LIN {X 0,Y 174.751,Z 590.29,A -85,B 0,C 180,E1 -20666.168,E2 -20666.168} C_VEL
LIN {X 0,Y 175.448,Z 592.178,A -85,B 0,C 180,E1 -20665.716,E2 -20665.716} C_VEL
LIN {X 0,Y 170.864,Z 646.273,A -85,B 0,C 180,E1 -20663.89,E2 -20663.89} C_VEL
LIN {X 0,Y 168.633,Z 660.424,A -85,B 0,C 180,E1 -20663.092,E2 -20663.092} C_VEL
LIN {X 0,Y 165.16,Z 674.762,A -85,B 0,C 180,E1 -20661.921,E2 -20661.921} C_VEL
LIN {X 0,Y 160.858,Z 688.251,A -85,B 0,C 180,E1 -20660.352,E2 -20660.352} C_VEL
LIN {X 0,Y 156.099,Z 700.216,A -85,B 0,C 180,E1 -20658.455,E2 -20658.455} C_VEL
LIN {X 0,Y 150.998,Z 711.144,A -85,B 0,C 180,E1 -20656.167,E2 -20656.167} C_VEL
LIN {X 0,Y 145.727,Z 721.318,A -85,B 0,C 180,E1 -20653.335,E2 -20653.335} C_VEL
LIN {X 0,Y 139.98,Z 731.094,A -85,B 0,C 180,E1 -20649.797,E2 -20649.797} C_VEL
LIN {X 0,Y 134.657,Z 739.228,A -85,B 0,C 180,E1 -20645.951,E2 -20645.951} C_VEL
LIN {X 0,Y 129.545,Z 746.964,A -85,B 0,C 180,E1 -20641.018,E2 -20641.018} C_VEL
LIN {X 0,Y 125.777,Z 752.256,A -85,B 0,C 180,E1 -20636.547,E2 -20636.547} C_VEL
LIN {X 0,Y 123.001,Z 756.514,A -85,B 0,C 180,E1 -20631.797,E2 -20631.797} C_VEL
LIN {X 0,Y 121.021,Z 759.832,A -85,B 0,C 180,E1 -20626.875,E2 -20626.875} C_VEL
LIN {X 0,Y 119.673,Z 762.879,A -85,B 0,C 180,E1 -20620.143,E2 -20620.143} C_VEL
LIN {X 0,Y 119.597,Z 764.442,A -85,B 0,C 180,E1 -20613.364,E2 -20613.364} C_VEL
LIN {X 0,Y 119.785,Z 764.659,A -85,B 0,C 180,E1 -20609.996,E2 -20609.996} C_VEL
LIN {X 0,Y 119.65,Z 764.459,A -85,B 0,C 180,E1 -20606.628,E2 -20606.628} C_VEL
LIN {X 0,Y 120.033,Z 762.933,A -85,B 0,C 180,E1 -20599.879,E2 -20599.879} C_VEL
LIN {X 0,Y 121.971,Z 759.942,A -85,B 0,C 180,E1 -20593.251,E2 -20593.251} C_VEL
LIN {X 0,Y 124.627,Z 756.694,A -85,B 0,C 180,E1 -20588.493,E2 -20588.493} C_VEL
LIN {X 0,Y 126.269,Z 755.1,A -85,B 0,C 180,E1 -20586.415,E2 -20586.415} C_VEL
LIN {X 0,Y 130.164,Z 758.008,A -85,B 0,C 180,E1 -20580.922,E2 -20580.922} C_VEL
LIN {X 0,Y 136.162,Z 760.226,A -85,B 0,C 180,E1 -20575.401,E2 -20575.401} C_VEL
LIN {X 0,Y 143.723,Z 761.469,A -85,B 0,C 180,E1 -20570.524,E2 -20570.524} C_VEL
LIN {X 0,Y 152.615,Z 761.755,A -85,B 0,C 180,E1 -20566.306,E2 -20566.306} C_VEL
LIN {X 0,Y 160.985,Z 761.235,A -85,B 0,C 180,E1 -20563.302,E2 -20563.302} C_VEL
LIN {X 0,Y 161.397,Z 761.087,A -85,B 0,C 180,E1 -20562.555,E2 -20562.555} C_VEL
LIN {X 0,Y 153.739,Z 760.626,A -85,B 0,C 180,E1 -20559.791,E2 -20559.791} C_VEL
LIN {X 0,Y 144.738,Z 758.979,A -85,B 0,C 180,E1 -20555.639,E2 -20555.639} C_VEL
LIN {X 0,Y 140.613,Z 757.696,A -85,B 0,C 180,E1 -20553.352,E2 -20553.352} C_VEL
LIN {X 0,Y 133.608,Z 754.257,A -85,B 0,C 180,E1 -20548.256,E2 -20548.256} C_VEL
LIN {X 0,Y 128.205,Z 749.58,A -85,B 0,C 180,E1 -20542.565,E2 -20542.565} C_VEL
LIN {X 0,Y 124.544,Z 743.565,A -85,B 0,C 180,E1 -20536.388,E2 -20536.388} C_VEL
LIN {X 0,Y 122.611,Z 737,A -85,B 0,C 180,E1 -20530.736,E2 -20530.736} C_VEL
LIN {X 0,Y 122.043,Z 729.036,A -85,B 0,C 180,E1 -20524.955,E2 -20524.955} C_VEL
LIN {X 0,Y 122.077,Z 720.491,A -85,B 0,C 180,E1 -20520,E2 -20520} C_VEL
LIN {X 0,Y 122.258,Z 711.841,A -85,B 0,C 180,E1 -20515.879,E2 -20515.879} C_VEL
LIN {X 0,Y 122.735,Z 702.53,A -85,B 0,C 180,E1 -20512.183,E2 -20512.183} C_VEL
LIN {X 0,Y 123.406,Z 691.305,A -85,B 0,C 180,E1 -20508.55,E2 -20508.55} C_VEL
LIN {X 0,Y 123.591,Z 689.165,A -85,B 0,C 180,E1 -20507.466,E2 -20507.466} C_VEL
LIN {X 0,Y 123.823,Z 687.977,A -85,B 0,C 180,E1 -20506.056,E2 -20506.056} C_VEL
LIN {X 0,Y 124.277,Z 687.395,A -85,B 0,C 180,E1 -20504.226,E2 -20504.226} C_VEL
LIN {X 0,Y 125.905,Z 686.979,A -85,B 0,C 180,E1 -20501.018,E2 -20501.018} C_VEL
LIN {X 0,Y 127.633,Z 685.962,A -85,B 0,C 180,E1 -20499.327,E2 -20499.327} C_VEL
LIN {X 0,Y 129.648,Z 684.696,A -85,B 0,C 180,E1 -20497.699,E2 -20497.699} C_VEL
LIN {X 0,Y 133.094,Z 681.626,A -85,B 0,C 180,E1 -20495.842,E2 -20495.842} C_VEL
LIN {X 0,Y 137.05,Z 677.069,A -85,B 0,C 180,E1 -20494.334,E2 -20494.334} C_VEL
LIN {X 0,Y 138.247,Z 675.526,A -85,B 0,C 180,E1 -20493.975,E2 -20493.975} C_VEL
LIN {X 0,Y 141.117,Z 673.06,A -85,B 0,C 180,E1 -20492.488,E2 -20492.488} C_VEL
LIN {X 0,Y 145.003,Z 668.739,A -85,B 0,C 180,E1 -20491.008,E2 -20491.008} C_VEL
LIN {X 0,Y 149.365,Z 662.342,A -85,B 0,C 180,E1 -20489.788,E2 -20489.788} C_VEL
LIN {X 0,Y 153.704,Z 653.819,A -85,B 0,C 180,E1 -20488.901,E2 -20488.901} C_VEL
LIN {X 0,Y 154.898,Z 651.2,A -85,B 0,C 180,E1 -20488.661,E2 -20488.661} C_VEL
LIN {X 0,Y 158.174,Z 646.403,A -85,B 0,C 180,E1 -20487.439,E2 -20487.439} C_VEL
LIN {X 0,Y 161.889,Z 638.911,A -85,B 0,C 180,E1 -20486.261,E2 -20486.261} C_VEL
LIN {X 0,Y 165.983,Z 627.33,A -85,B 0,C 180,E1 -20485.022,E2 -20485.022} C_VEL
LIN {X 0,Y 169.425,Z 615.622,A -85,B 0,C 180,E1 -20484.131,E2 -20484.131} C_VEL
LIN {X 0,Y 167.38,Z 640.416,A -85,B 0,C 180,E1 -20483.235,E2 -20483.235} C_VEL
LIN {X 0,Y 165.141,Z 654.079,A -85,B 0,C 180,E1 -20482.437,E2 -20482.437} C_VEL
LIN {X 0,Y 162.14,Z 666.874,A -85,B 0,C 180,E1 -20481.285,E2 -20481.285} C_VEL
LIN {X 0,Y 157.903,Z 680.096,A -85,B 0,C 180,E1 -20479.664,E2 -20479.664} C_VEL
LIN {X 0,Y 153.219,Z 691.732,A -85,B 0,C 180,E1 -20477.705,E2 -20477.705} C_VEL
LIN {X 0,Y 148.082,Z 702.301,A -85,B 0,C 180,E1 -20475.394,E2 -20475.394} C_VEL
LIN {X 0,Y 142.637,Z 712.201,A -85,B 0,C 180,E1 -20472.492,E2 -20472.492} C_VEL
LIN {X 0,Y 136.949,Z 721.337,A -85,B 0,C 180,E1 -20468.955,E2 -20468.955} C_VEL
LIN {X 0,Y 131.412,Z 728.995,A -85,B 0,C 180,E1 -20465.098,E2 -20465.098} C_VEL
LIN {X 0,Y 125.818,Z 736.115,A -85,B 0,C 180,E1 -20460.185,E2 -20460.185} C_VEL
LIN {X 0,Y 121.759,Z 740.971,A -85,B 0,C 180,E1 -20455.657,E2 -20455.657} C_VEL
LIN {X 0,Y 118.435,Z 744.801,A -85,B 0,C 180,E1 -20450.862,E2 -20450.862} C_VEL
LIN {X 0,Y 115.262,Z 748.408,A -85,B 0,C 180,E1 -20444.121,E2 -20444.121} C_VEL
LIN {X 0,Y 113.482,Z 750.529,A -85,B 0,C 180,E1 -20437.12,E2 -20437.12} C_VEL
LIN {X 0,Y 112.893,Z 751.232,A -85,B 0,C 180,E1 -20430.005,E2 -20430.005} C_VEL
LIN {X 0,Y 113.479,Z 750.486,A -85,B 0,C 180,E1 -20422.89,E2 -20422.89} C_VEL
LIN {X 0,Y 115.257,Z 748.33,A -85,B 0,C 180,E1 -20415.888,E2 -20415.888} C_VEL
LIN {X 0,Y 118.436,Z 744.678,A -85,B 0,C 180,E1 -20409.148,E2 -20409.148} C_VEL
LIN {X 0,Y 121.806,Z 740.807,A -85,B 0,C 180,E1 -20404.364,E2 -20404.364} C_VEL
LIN {X 0,Y 125.949,Z 735.902,A -85,B 0,C 180,E1 -20399.859,E2 -20399.859} C_VEL
LIN {X 0,Y 130.592,Z 729.843,A -85,B 0,C 180,E1 -20395.598,E2 -20395.598} C_VEL
LIN {X 0,Y 136.018,Z 722.398,A -85,B 0,C 180,E1 -20391.687,E2 -20391.687} C_VEL
LIN {X 0,Y 141.435,Z 713.947,A -85,B 0,C 180,E1 -20388.264,E2 -20388.264} C_VEL
LIN {X 0,Y 147.09,Z 703.928,A -85,B 0,C 180,E1 -20385.195,E2 -20385.195} C_VEL
LIN {X 0,Y 152.145,Z 693.71,A -85,B 0,C 180,E1 -20382.841,E2 -20382.841} C_VEL
LIN {X 0,Y 156.789,Z 682.529,A -85,B 0,C 180,E1 -20380.857,E2 -20380.857} C_VEL
LIN {X 0,Y 160.982,Z 670.126,A -85,B 0,C 180,E1 -20379.209,E2 -20379.209} C_VEL
LIN {X 0,Y 164.303,Z 657.215,A -85,B 0,C 180,E1 -20377.946,E2 -20377.946} C_VEL
LIN {X 0,Y 166.571,Z 644.664,A -85,B 0,C 180,E1 -20377.095,E2 -20377.095} C_VEL
LIN {X 0,Y 168.055,Z 630.758,A -85,B 0,C 180,E1 -20376.513,E2 -20376.513} C_VEL
LIN {X 0,Y 171.047,Z 593.041,A -85,B 0,C 180,E1 -20375.296,E2 -20375.296} C_VEL
LIN {X 0,Y 167.73,Z 584.739,A -85,B 0,C 180,E1 -20372.916,E2 -20372.916} C_VEL
LIN {X 0,Y 163.421,Z 575.531,A -85,B 0,C 180,E1 -20369.525,E2 -20369.525} C_VEL
LIN {X 0,Y 160.098,Z 569.15,A -85,B 0,C 180,E1 -20366.549,E2 -20366.549} C_VEL
LIN {X 0,Y 156.776,Z 563.254,A -85,B 0,C 180,E1 -20363.109,E2 -20363.109} C_VEL
LIN {X 0,Y 153.307,Z 557.682,A -85,B 0,C 180,E1 -20358.718,E2 -20358.718} C_VEL
LIN {X 0,Y 150.18,Z 552.762,A -85,B 0,C 180,E1 -20353.188,E2 -20353.188} C_VEL
LIN {X 0,Y 147.985,Z 549.73,A -85,B 0,C 180,E1 -20346.3,E2 -20346.3} C_VEL
LIN {X 0,Y 147.618,Z 548.691,A -85,B 0,C 180,E1 -20341.345,E2 -20341.345} C_VEL
LIN {X 0,Y 147.76,Z 549.144,A -85,B 0,C 180,E1 -20338.638,E2 -20338.638} C_VEL
LIN {X 0,Y 149.497,Z 552.083,A -85,B 0,C 180,E1 -20331.538,E2 -20331.538} C_VEL
LIN {X 0,Y 150.744,Z 553.976,A -85,B 0,C 180,E1 -20328.742,E2 -20328.742} C_VEL
LIN {X 0,Y 154.198,Z 559.575,A -85,B 0,C 180,E1 -20323.149,E2 -20323.149} C_VEL
LIN {X 0,Y 157.289,Z 564.846,A -85,B 0,C 180,E1 -20319.38,E2 -20319.38} C_VEL
LIN {X 0,Y 160.115,Z 570.007,A -85,B 0,C 180,E1 -20316.475,E2 -20316.475} C_VEL
LIN {X 0,Y 163.501,Z 576.58,A -85,B 0,C 180,E1 -20313.429,E2 -20313.429} C_VEL
LIN {X 0,Y 167.808,Z 586.127,A -85,B 0,C 180,E1 -20310.003,E2 -20310.003} C_VEL
LIN {X 0,Y 171.157,Z 594.739,A -85,B 0,C 180,E1 -20307.564,E2 -20307.564} C_VEL
LIN {X 0,Y 166.751,Z 645.455,A -85,B 0,C 180,E1 -20305.842,E2 -20305.842} C_VEL
LIN {X 0,Y 164.492,Z 659.477,A -85,B 0,C 180,E1 -20305.092,E2 -20305.092} C_VEL
LIN {X 0,Y 161.167,Z 673,A -85,B 0,C 180,E1 -20304.036,E2 -20304.036} C_VEL
LIN {X 0,Y 157.033,Z 685.93,A -85,B 0,C 180,E1 -20302.592,E2 -20302.592} C_VEL
LIN {X 0,Y 152.067,Z 698.358,A -85,B 0,C 180,E1 -20300.72,E2 -20300.72} C_VEL
LIN {X 0,Y 146.705,Z 709.591,A -85,B 0,C 180,E1 -20298.457,E2 -20298.457} C_VEL
LIN {X 0,Y 141.085,Z 720.013,A -85,B 0,C 180,E1 -20295.62,E2 -20295.62} C_VEL
LIN {X 0,Y 135.553,Z 729.147,A -85,B 0,C 180,E1 -20292.371,E2 -20292.371} C_VEL
LIN {X 0,Y 129.818,Z 737.545,A -85,B 0,C 180,E1 -20288.499,E2 -20288.499} C_VEL
LIN {X 0,Y 124.139,Z 745.513,A -85,B 0,C 180,E1 -20283.498,E2 -20283.498} C_VEL
LIN {X 0,Y 119.214,Z 752.093,A -85,B 0,C 180,E1 -20277.836,E2 -20277.836} C_VEL
LIN {X 0,Y 115.577,Z 757.318,A -85,B 0,C 180,E1 -20271.393,E2 -20271.393} C_VEL
LIN {X 0,Y 113.214,Z 761.13,A -85,B 0,C 180,E1 -20264.373,E2 -20264.373} C_VEL
LIN {X 0,Y 112.407,Z 763.432,A -85,B 0,C 180,E1 -20257.179,E2 -20257.179} C_VEL
LIN {X 0,Y 112.541,Z 764.134,A -85,B 0,C 180,E1 -20252.333,E2 -20252.333} C_VEL
LIN {X 0,Y 112.691,Z 764.25,A -85,B 0,C 180,E1 -20249.995,E2 -20249.995} C_VEL
LIN {X 0,Y 112.555,Z 764.049,A -85,B 0,C 180,E1 -20246.415,E2 -20246.415} C_VEL
LIN {X 0,Y 112.66,Z 763.47,A -85,B 0,C 180,E1 -20242.828,E2 -20242.828} C_VEL
LIN {X 0,Y 113.903,Z 761.214,A -85,B 0,C 180,E1 -20235.707,E2 -20235.707} C_VEL
LIN {X 0,Y 116.945,Z 757.47,A -85,B 0,C 180,E1 -20228.86,E2 -20228.86} C_VEL
LIN {X 0,Y 120.851,Z 753.596,A -85,B 0,C 180,E1 -20223.905,E2 -20223.905} C_VEL
LIN {X 0,Y 127.135,Z 757.49,A -85,B 0,C 180,E1 -20216.436,E2 -20216.436} C_VEL
LIN {X 0,Y 134.293,Z 759.63,A -85,B 0,C 180,E1 -20211.093,E2 -20211.093} C_VEL
LIN {X 0,Y 142.821,Z 760.817,A -85,B 0,C 180,E1 -20206.451,E2 -20206.451} C_VEL
LIN {X 0,Y 150.668,Z 761.111,A -85,B 0,C 180,E1 -20203.268,E2 -20203.268} C_VEL
LIN {X 0,Y 150.095,Z 760.873,A -85,B 0,C 180,E1 -20202.206,E2 -20202.206} C_VEL
LIN {X 0,Y 143.541,Z 759.697,A -85,B 0,C 180,E1 -20199.531,E2 -20199.531} C_VEL
LIN {X 0,Y 134.792,Z 756.968,A -85,B 0,C 180,E1 -20194.997,E2 -20194.997} C_VEL
LIN {X 0,Y 127.504,Z 753.065,A -85,B 0,C 180,E1 -20189.741,E2 -20189.741} C_VEL
LIN {X 0,Y 121.857,Z 747.927,A -85,B 0,C 180,E1 -20183.811,E2 -20183.811} C_VEL
LIN {X 0,Y 118.049,Z 741.477,A -85,B 0,C 180,E1 -20177.317,E2 -20177.317} C_VEL
LIN {X 0,Y 115.897,Z 733.429,A -85,B 0,C 180,E1 -20170.481,E2 -20170.481} C_VEL
LIN {X 0,Y 115.491,Z 726.032,A -85,B 0,C 180,E1 -20165.237,E2 -20165.237} C_VEL
LIN {X 0,Y 115.449,Z 718.689,A -85,B 0,C 180,E1 -20160.871,E2 -20160.871} C_VEL
LIN {X 0,Y 115.657,Z 708.699,A -85,B 0,C 180,E1 -20156.08,E2 -20156.08} C_VEL
LIN {X 0,Y 116.092,Z 698.828,A -85,B 0,C 180,E1 -20152.171,E2 -20152.171} C_VEL
LIN {X 0,Y 116.215,Z 695.374,A -85,B 0,C 180,E1 -20150.92,E2 -20150.92} C_VEL
LIN {X 0,Y 115.98,Z 695.896,A -85,B 0,C 180,E1 -20150.407,E2 -20150.407} C_VEL
LIN {X 0,Y 116.047,Z 696.135,A -85,B 0,C 180,E1 -20149.532,E2 -20149.532} C_VEL
LIN {X 0,Y 117.022,Z 695.467,A -85,B 0,C 180,E1 -20147.865,E2 -20147.865} C_VEL
LIN {X 0,Y 120.501,Z 692.137,A -85,B 0,C 180,E1 -20144.784,E2 -20144.784} C_VEL
LIN {X 0,Y 123.407,Z 690.151,A -85,B 0,C 180,E1 -20141.746,E2 -20141.746} C_VEL
LIN {X 0,Y 125.691,Z 687.944,A -85,B 0,C 180,E1 -20140.397,E2 -20140.397} C_VEL
LIN {X 0,Y 127.127,Z 686.36,A -85,B 0,C 180,E1 -20139.702,E2 -20139.702} C_VEL
LIN {X 0,Y 127.633,Z 685.962,A -85,B 0,C 180,E1 -20139.327,E2 -20139.327} C_VEL
LIN {X 0,Y 130.12,Z 684.459,A -85,B 0,C 180,E1 -20137.326,E2 -20137.326} C_VEL
LIN {X 0,Y 135.875,Z 682.058,A -85,B 0,C 180,E1 -20132.88,E2 -20132.88} C_VEL
LIN {X 0,Y 138.121,Z 680.497,A -85,B 0,C 180,E1 -20131.678,E2 -20131.678} C_VEL
LIN {X 0,Y 142.493,Z 676.654,A -85,B 0,C 180,E1 -20129.897,E2 -20129.897} C_VEL
LIN {X 0,Y 145.897,Z 673.011,A -85,B 0,C 180,E1 -20128.812,E2 -20128.812} C_VEL
LIN {X 0,Y 150.887,Z 666.322,A -85,B 0,C 180,E1 -20127.613,E2 -20127.613} C_VEL
LIN {X 0,Y 155.631,Z 657.999,A -85,B 0,C 180,E1 -20126.796,E2 -20126.796} C_VEL
LIN {X 0,Y 157.05,Z 655.124,A -85,B 0,C 180,E1 -20126.542,E2 -20126.542} C_VEL
LIN {X 0,Y 160.655,Z 649.982,A -85,B 0,C 180,E1 -20125.432,E2 -20125.432} C_VEL
LIN {X 0,Y 162.342,Z 647.1,A -85,B 0,C 180,E1 -20124.961,E2 -20124.961} C_VEL
LIN {X 0,Y 159.457,Z 661.267,A -85,B 0,C 180,E1 -20123.903,E2 -20123.903} C_VEL
LIN {X 0,Y 155.953,Z 673.577,A -85,B 0,C 180,E1 -20122.591,E2 -20122.591} C_VEL
LIN {X 0,Y 151.65,Z 685.301,A -85,B 0,C 180,E1 -20120.924,E2 -20120.924} C_VEL
LIN {X 0,Y 146.125,Z 697.171,A -85,B 0,C 180,E1 -20118.725,E2 -20118.725} C_VEL
LIN {X 0,Y 140.912,Z 706.825,A -85,B 0,C 180,E1 -20116.323,E2 -20116.323} C_VEL
LIN {X 0,Y 135.252,Z 716.191,A -85,B 0,C 180,E1 -20113.203,E2 -20113.203} C_VEL
LIN {X 0,Y 129.513,Z 724.461,A -85,B 0,C 180,E1 -20109.619,E2 -20109.619} C_VEL
LIN {X 0,Y 123.922,Z 731.606,A -85,B 0,C 180,E1 -20105.547,E2 -20105.547} C_VEL
LIN {X 0,Y 118.24,Z 738.292,A -85,B 0,C 180,E1 -20100.351,E2 -20100.351} C_VEL
LIN {X 0,Y 114.142,Z 742.772,A -85,B 0,C 180,E1 -20095.536,E2 -20095.536} C_VEL
LIN {X 0,Y 111.84,Z 745.21,A -85,B 0,C 180,E1 -20092.155,E2 -20092.155} C_VEL
LIN {X 0,Y 108.391,Z 748.817,A -85,B 0,C 180,E1 -20085.037,E2 -20085.037} C_VEL
LIN {X 0,Y 106.463,Z 750.937,A -85,B 0,C 180,E1 -20077.592,E2 -20077.592} C_VEL
LIN {X 0,Y 105.824,Z 751.64,A -85,B 0,C 180,E1 -20070.005,E2 -20070.005} C_VEL
LIN {X 0,Y 106.461,Z 750.894,A -85,B 0,C 180,E1 -20062.418,E2 -20062.418} C_VEL
LIN {X 0,Y 108.385,Z 748.74,A -85,B 0,C 180,E1 -20054.972,E2 -20054.972} C_VEL
LIN {X 0,Y 111.841,Z 745.089,A -85,B 0,C 180,E1 -20047.855,E2 -20047.855} C_VEL
LIN {X 0,Y 115.461,Z 741.218,A -85,B 0,C 180,E1 -20042.843,E2 -20042.843} C_VEL
LIN {X 0,Y 119.858,Z 736.318,A -85,B 0,C 180,E1 -20038.154,E2 -20038.154} C_VEL
LIN {X 0,Y 124.818,Z 730.262,A -85,B 0,C 180,E1 -20033.762,E2 -20033.762} C_VEL
LIN {X 0,Y 130.541,Z 722.824,A -85,B 0,C 180,E1 -20029.761,E2 -20029.761} C_VEL
LIN {X 0,Y 136.559,Z 713.876,A -85,B 0,C 180,E1 -20026.097,E2 -20026.097} C_VEL
LIN {X 0,Y 142.147,Z 704.392,A -85,B 0,C 180,E1 -20023.181,E2 -20023.181} C_VEL
LIN {X 0,Y 147.434,Z 694.197,A -85,B 0,C 180,E1 -20020.828,E2 -20020.828} C_VEL
LIN {X 0,Y 152.259,Z 683.054,A -85,B 0,C 180,E1 -20018.845,E2 -20018.845} C_VEL
LIN {X 0,Y 156.615,Z 670.711,A -85,B 0,C 180,E1 -20017.207,E2 -20017.207} C_VEL
LIN {X 0,Y 160.061,Z 657.901,A -85,B 0,C 180,E1 -20015.954,E2 -20015.954} C_VEL
LIN {X 0,Y 162.412,Z 645.601,A -85,B 0,C 180,E1 -20015.109,E2 -20015.109} C_VEL
LIN {X 0,Y 163.958,Z 632.23,A -85,B 0,C 180,E1 -20014.533,E2 -20014.533} C_VEL
LIN {X 0,Y 166.984,Z 595.617,A -85,B 0,C 180,E1 -20013.352,E2 -20013.352} C_VEL
LIN {X 0,Y 163.154,Z 586.222,A -85,B 0,C 180,E1 -20010.301,E2 -20010.301} C_VEL
LIN {X 0,Y 159.55,Z 578.432,A -85,B 0,C 180,E1 -20007.075,E2 -20007.075} C_VEL
LIN {X 0,Y 156.34,Z 572.241,A -85,B 0,C 180,E1 -20003.779,E2 -20003.779} C_VEL
LIN {X 0,Y 153.865,Z 567.749,A -85,B 0,C 180,E1 -20000.803,E2 -20000.803} C_VEL
LIN {X 0,Y 151.679,Z 564.144,A -85,B 0,C 180,E1 -19997.703,E2 -19997.703} C_VEL
LIN {X 0,Y 149.018,Z 559.587,A -85,B 0,C 180,E1 -19992.599,E2 -19992.599} C_VEL
LIN {X 0,Y 147.106,Z 556.814,A -85,B 0,C 180,E1 -19986.258,E2 -19986.258} C_VEL
LIN {X 0,Y 146.748,Z 556.001,A -85,B 0,C 180,E1 -19982.745,E2 -19982.745} C_VEL
LIN {X 0,Y 146.814,Z 555.905,A -85,B 0,C 180,E1 -19979.658,E2 -19979.658} C_VEL
LIN {X 0,Y 148.364,Z 558.901,A -85,B 0,C 180,E1 -19972.173,E2 -19972.173} C_VEL
LIN {X 0,Y 149.535,Z 560.838,A -85,B 0,C 180,E1 -19969.336,E2 -19969.336} C_VEL
LIN {X 0,Y 152.627,Z 566.192,A -85,B 0,C 180,E1 -19963.962,E2 -19963.962} C_VEL
LIN {X 0,Y 155.328,Z 571.036,A -85,B 0,C 180,E1 -19960.422,E2 -19960.422} C_VEL
LIN {X 0,Y 158.322,Z 576.818,A -85,B 0,C 180,E1 -19957.144,E2 -19957.144} C_VEL
LIN {X 0,Y 161.296,Z 583.175,A -85,B 0,C 180,E1 -19954.285,E2 -19954.285} C_VEL
LIN {X 0,Y 164.848,Z 591.51,A -85,B 0,C 180,E1 -19951.25,E2 -19951.25} C_VEL
LIN {X 0,Y 167.045,Z 597.374,A -85,B 0,C 180,E1 -19949.503,E2 -19949.503} C_VEL
LIN {X 0,Y 162.682,Z 645.77,A -85,B 0,C 180,E1 -19947.858,E2 -19947.858} C_VEL
LIN {X 0,Y 160.301,Z 659.728,A -85,B 0,C 180,E1 -19947.108,E2 -19947.108} C_VEL
LIN {X 0,Y 156.757,Z 673.502,A -85,B 0,C 180,E1 -19946.033,E2 -19946.033} C_VEL
LIN {X 0,Y 152.808,Z 685.375,A -85,B 0,C 180,E1 -19944.716,E2 -19944.716} C_VEL
LIN {X 0,Y 147.658,Z 697.849,A -85,B 0,C 180,E1 -19942.861,E2 -19942.861} C_VEL
LIN {X 0,Y 142.094,Z 709.123,A -85,B 0,C 180,E1 -19940.601,E2 -19940.601} C_VEL
LIN {X 0,Y 136.6,Z 718.82,A -85,B 0,C 180,E1 -19938.023,E2 -19938.023} C_VEL
LIN {X 0,Y 130.345,Z 728.71,A -85,B 0,C 180,E1 -19934.496,E2 -19934.496} C_VEL
LIN {X 0,Y 124.307,Z 737.117,A -85,B 0,C 180,E1 -19930.549,E2 -19930.549} C_VEL
LIN {X 0,Y 118.219,Z 745.089,A -85,B 0,C 180,E1 -19925.418,E2 -19925.418} C_VEL
LIN {X 0,Y 113.151,Z 751.418,A -85,B 0,C 180,E1 -19919.789,E2 -19919.789} C_VEL
LIN {X 0,Y 109.799,Z 755.68,A -85,B 0,C 180,E1 -19914.58,E2 -19914.58} C_VEL
LIN {X 0,Y 107.391,Z 759.003,A -85,B 0,C 180,E1 -19909.095,E2 -19909.095} C_VEL
LIN {X 0,Y 105.623,Z 762.053,A -85,B 0,C 180,E1 -19901.509,E2 -19901.509} C_VEL
LIN {X 0,Y 105.391,Z 763.62,A -85,B 0,C 180,E1 -19893.819,E2 -19893.819} C_VEL
LIN {X 0,Y 105.597,Z 763.84,A -85,B 0,C 180,E1 -19889.995,E2 -19889.995} C_VEL
LIN {X 0,Y 105.463,Z 763.639,A -85,B 0,C 180,E1 -19886.174,E2 -19886.174} C_VEL
LIN {X 0,Y 105.606,Z 763.06,A -85,B 0,C 180,E1 -19882.346,E2 -19882.346} C_VEL
LIN {X 0,Y 107.01,Z 760.803,A -85,B 0,C 180,E1 -19874.764,E2 -19874.764} C_VEL
LIN {X 0,Y 110.344,Z 757.059,A -85,B 0,C 180,E1 -19867.528,E2 -19867.528} C_VEL
LIN {X 0,Y 115.494,Z 752.104,A -85,B 0,C 180,E1 -19861.361,E2 -19861.361} C_VEL
LIN {X 0,Y 115.877,Z 752.058,A -85,B 0,C 180,E1 -19860.969,E2 -19860.969} C_VEL
LIN {X 0,Y 121.511,Z 755.529,A -85,B 0,C 180,E1 -19854.658,E2 -19854.658} C_VEL
LIN {X 0,Y 128.981,Z 758.069,A -85,B 0,C 180,E1 -19849.162,E2 -19849.162} C_VEL
LIN {X 0,Y 139.647,Z 759.866,A -85,B 0,C 180,E1 -19843.665,E2 -19843.665} C_VEL
LIN {X 0,Y 140.607,Z 759.968,A -85,B 0,C 180,E1 -19843.271,E2 -19843.271} C_VEL
LIN {X 0,Y 139.919,Z 759.638,A -85,B 0,C 180,E1 -19842.147,E2 -19842.147} C_VEL
LIN {X 0,Y 133.521,Z 757.741,A -85,B 0,C 180,E1 -19839.17,E2 -19839.17} C_VEL
LIN {X 0,Y 125.179,Z 753.97,A -85,B 0,C 180,E1 -19834.155,E2 -19834.155} C_VEL
LIN {X 0,Y 118.379,Z 749.006,A -85,B 0,C 180,E1 -19828.356,E2 -19828.356} C_VEL
LIN {X 0,Y 113.418,Z 742.771,A -85,B 0,C 180,E1 -19821.826,E2 -19821.826} C_VEL
LIN {X 0,Y 110.584,Z 736.136,A -85,B 0,C 180,E1 -19815.67,E2 -19815.67} C_VEL
LIN {X 0,Y 109.179,Z 726.907,A -85,B 0,C 180,E1 -19808.327,E2 -19808.327} C_VEL
LIN {X 0,Y 108.962,Z 718.206,A -85,B 0,C 180,E1 -19802.772,E2 -19802.772} C_VEL
LIN {X 0,Y 109.001,Z 709.366,A -85,B 0,C 180,E1 -19798.152,E2 -19798.152} C_VEL
LIN {X 0,Y 109.105,Z 704.328,A -85,B 0,C 180,E1 -19795.844,E2 -19795.844} C_VEL
LIN {X 0,Y 108.732,Z 704.907,A -85,B 0,C 180,E1 -19794.436,E2 -19794.436} C_VEL
LIN {X 0,Y 109.327,Z 704.436,A -85,B 0,C 180,E1 -19792.613,E2 -19792.613} C_VEL
LIN {X 0,Y 111.986,Z 701.907,A -85,B 0,C 180,E1 -19789.147,E2 -19789.147} C_VEL
LIN {X 0,Y 114.256,Z 700.43,A -85,B 0,C 180,E1 -19785.756,E2 -19785.756} C_VEL
LIN {X 0,Y 117.495,Z 697.696,A -85,B 0,C 180,E1 -19783.159,E2 -19783.159} C_VEL
LIN {X 0,Y 121.319,Z 695.24,A -85,B 0,C 180,E1 -19779.66,E2 -19779.66} C_VEL
LIN {X 0,Y 126.155,Z 691.085,A -85,B 0,C 180,E1 -19777.047,E2 -19777.047} C_VEL
LIN {X 0,Y 128.083,Z 689.921,A -85,B 0,C 180,E1 -19775.698,E2 -19775.698} C_VEL
LIN {X 0,Y 132.275,Z 686.527,A -85,B 0,C 180,E1 -19773.668,E2 -19773.668} C_VEL
LIN {X 0,Y 136.085,Z 682.702,A -85,B 0,C 180,E1 -19772.302,E2 -19772.302} C_VEL
LIN {X 0,Y 138.121,Z 680.497,A -85,B 0,C 180,E1 -19771.678,E2 -19771.678} C_VEL
LIN {X 0,Y 141.302,Z 678.49,A -85,B 0,C 180,E1 -19770.035,E2 -19770.035} C_VEL
LIN {X 0,Y 146.87,Z 675.936,A -85,B 0,C 180,E1 -19767.119,E2 -19767.119} C_VEL
LIN {X 0,Y 149.751,Z 673.72,A -85,B 0,C 180,E1 -19766.042,E2 -19766.042} C_VEL
LIN {X 0,Y 150.936,Z 672.387,A -85,B 0,C 180,E1 -19765.742,E2 -19765.742} C_VEL
LIN {X 0,Y 152.462,Z 670.362,A -85,B 0,C 180,E1 -19765.463,E2 -19765.463} C_VEL
LIN {X 0,Y 152.39,Z 672.172,A -85,B 0,C 180,E1 -19764.95,E2 -19764.95} C_VEL
LIN {X 0,Y 147.914,Z 684.265,A -85,B 0,C 180,E1 -19763.307,E2 -19763.307} C_VEL
LIN {X 0,Y 142.819,Z 695.255,A -85,B 0,C 180,E1 -19761.375,E2 -19761.375} C_VEL
LIN {X 0,Y 137.323,Z 705.322,A -85,B 0,C 180,E1 -19759.021,E2 -19759.021} C_VEL
LIN {X 0,Y 131.379,Z 714.847,A -85,B 0,C 180,E1 -19756.018,E2 -19756.018} C_VEL
LIN {X 0,Y 125.18,Z 723.549,A -85,B 0,C 180,E1 -19752.36,E2 -19752.36} C_VEL
LIN {X 0,Y 119.138,Z 730.928,A -85,B 0,C 180,E1 -19748.277,E2 -19748.277} C_VEL
LIN {X 0,Y 113.767,Z 736.941,A -85,B 0,C 180,E1 -19743.783,E2 -19743.783} C_VEL
LIN {X 0,Y 109.17,Z 741.79,A -85,B 0,C 180,E1 -19738.875,E2 -19738.875} C_VEL
LIN {X 0,Y 105.317,Z 745.618,A -85,B 0,C 180,E1 -19733.608,E2 -19733.608} C_VEL
LIN {X 0,Y 101.569,Z 749.225,A -85,B 0,C 180,E1 -19726.073,E2 -19726.073} C_VEL
LIN {X 0,Y 99.438,Z 751.346,A -85,B 0,C 180,E1 -19718.131,E2 -19718.131} C_VEL
LIN {X 0,Y 98.736,Z 752.049,A -85,B 0,C 180,E1 -19710.005,E2 -19710.005} C_VEL
LIN {X 0,Y 99.434,Z 751.304,A -85,B 0,C 180,E1 -19701.879,E2 -19701.879} C_VEL
LIN {X 0,Y 101.563,Z 749.149,A -85,B 0,C 180,E1 -19693.937,E2 -19693.937} C_VEL
LIN {X 0,Y 105.317,Z 745.499,A -85,B 0,C 180,E1 -19686.403,E2 -19686.403} C_VEL
LIN {X 0,Y 109.211,Z 741.629,A -85,B 0,C 180,E1 -19681.148,E2 -19681.148} C_VEL
LIN {X 0,Y 113.886,Z 736.734,A -85,B 0,C 180,E1 -19676.268,E2 -19676.268} C_VEL
LIN {X 0,Y 119.186,Z 730.681,A -85,B 0,C 180,E1 -19671.752,E2 -19671.752} C_VEL
LIN {X 0,Y 125.213,Z 723.251,A -85,B 0,C 180,E1 -19667.665,E2 -19667.665} C_VEL
LIN {X 0,Y 131.675,Z 714.102,A -85,B 0,C 180,E1 -19663.875,E2 -19663.875} C_VEL
LIN {X 0,Y 138.001,Z 703.795,A -85,B 0,C 180,E1 -19660.759,E2 -19660.759} C_VEL
LIN {X 0,Y 143.531,Z 693.404,A -85,B 0,C 180,E1 -19658.43,E2 -19658.43} C_VEL
LIN {X 0,Y 148.589,Z 682.005,A -85,B 0,C 180,E1 -19656.486,E2 -19656.486} C_VEL
LIN {X 0,Y 153.107,Z 669.308,A -85,B 0,C 180,E1 -19654.871,E2 -19654.871} C_VEL
LIN {X 0,Y 156.579,Z 656.024,A -85,B 0,C 180,E1 -19653.638,E2 -19653.638} C_VEL
LIN {X 0,Y 159.071,Z 642.186,A -85,B 0,C 180,E1 -19652.79,E2 -19652.79} C_VEL
LIN {X 0,Y 161.35,Z 619.119,A -85,B 0,C 180,E1 -19652.003,E2 -19652.003} C_VEL
LIN {X 0,Y 163.093,Z 598.441,A -85,B 0,C 180,E1 -19651.319,E2 -19651.319} C_VEL
LIN {X 0,Y 159.218,Z 588.732,A -85,B 0,C 180,E1 -19647.854,E2 -19647.854} C_VEL
LIN {X 0,Y 156.05,Z 581.76,A -85,B 0,C 180,E1 -19644.62,E2 -19644.62} C_VEL
LIN {X 0,Y 153.734,Z 577.167,A -85,B 0,C 180,E1 -19641.918,E2 -19641.918} C_VEL
LIN {X 0,Y 151.955,Z 573.777,A -85,B 0,C 180,E1 -19639.537,E2 -19639.537} C_VEL
LIN {X 0,Y 150.205,Z 570.703,A -85,B 0,C 180,E1 -19636.829,E2 -19636.829} C_VEL
LIN {X 0,Y 147.871,Z 566.432,A -85,B 0,C 180,E1 -19632.002,E2 -19632.002} C_VEL
LIN {X 0,Y 146.116,Z 563.7,A -85,B 0,C 180,E1 -19625.521,E2 -19625.521} C_VEL
LIN {X 0,Y 145.879,Z 563.086,A -85,B 0,C 180,E1 -19622.762,E2 -19622.762} C_VEL
LIN {X 0,Y 145.943,Z 563.002,A -85,B 0,C 180,E1 -19619.656,E2 -19619.656} C_VEL
LIN {X 0,Y 147.256,Z 565.724,A -85,B 0,C 180,E1 -19612.803,E2 -19612.803} C_VEL
LIN {X 0,Y 148.273,Z 567.537,A -85,B 0,C 180,E1 -19610.108,E2 -19610.108} C_VEL
LIN {X 0,Y 151.117,Z 572.839,A -85,B 0,C 180,E1 -19604.749,E2 -19604.749} C_VEL
LIN {X 0,Y 153.432,Z 577.289,A -85,B 0,C 180,E1 -19601.472,E2 -19601.472} C_VEL
LIN {X 0,Y 156.12,Z 582.807,A -85,B 0,C 180,E1 -19598.286,E2 -19598.286} C_VEL
LIN {X 0,Y 158.958,Z 589.288,A -85,B 0,C 180,E1 -19595.338,E2 -19595.338} C_VEL
LIN {X 0,Y 162.134,Z 597.32,A -85,B 0,C 180,E1 -19592.402,E2 -19592.402} C_VEL
LIN {X 0,Y 163.163,Z 600.213,A -85,B 0,C 180,E1 -19591.503,E2 -19591.503} C_VEL
LIN {X 0,Y 158.816,Z 646.037,A -85,B 0,C 180,E1 -19589.977,E2 -19589.977} C_VEL
LIN {X 0,Y 156.243,Z 660.344,A -85,B 0,C 180,E1 -19589.202,E2 -19589.202} C_VEL
LIN {X 0,Y 152.551,Z 674.005,A -85,B 0,C 180,E1 -19588.14,E2 -19588.14} C_VEL
LIN {X 0,Y 148.13,Z 686.593,A -85,B 0,C 180,E1 -19586.735,E2 -19586.735} C_VEL
LIN {X 0,Y 142.821,Z 698.741,A -85,B 0,C 180,E1 -19584.887,E2 -19584.887} C_VEL
LIN {X 0,Y 137.038,Z 709.745,A -85,B 0,C 180,E1 -19582.64,E2 -19582.64} C_VEL
LIN {X 0,Y 130.475,Z 720.681,A -85,B 0,C 180,E1 -19579.567,E2 -19579.567} C_VEL
LIN {X 0,Y 124.266,Z 729.783,A -85,B 0,C 180,E1 -19576.138,E2 -19576.138} C_VEL
LIN {X 0,Y 117.962,Z 737.943,A -85,B 0,C 180,E1 -19572.081,E2 -19572.081} C_VEL
LIN {X 0,Y 111.613,Z 745.693,A -85,B 0,C 180,E1 -19566.734,E2 -19566.734} C_VEL
LIN {X 0,Y 106.014,Z 752.067,A -85,B 0,C 180,E1 -19560.48,E2 -19560.48} C_VEL
LIN {X 0,Y 102.322,Z 756.484,A -85,B 0,C 180,E1 -19554.332,E2 -19554.332} C_VEL
LIN {X 0,Y 99.418,Z 760.302,A -85,B 0,C 180,E1 -19546.42,E2 -19546.42} C_VEL
LIN {X 0,Y 98.258,Z 762.607,A -85,B 0,C 180,E1 -19538.219,E2 -19538.219} C_VEL
LIN {X 0,Y 98.418,Z 763.376,A -85,B 0,C 180,E1 -19531.33,E2 -19531.33} C_VEL
LIN {X 0,Y 98.429,Z 763.371,A -85,B 0,C 180,E1 -19528.411,E2 -19528.411} C_VEL
LIN {X 0,Y 98.551,Z 762.649,A -85,B 0,C 180,E1 -19521.795,E2 -19521.795} C_VEL
LIN {X 0,Y 100.161,Z 760.393,A -85,B 0,C 180,E1 -19513.695,E2 -19513.695} C_VEL
LIN {X 0,Y 103.812,Z 756.649,A -85,B 0,C 180,E1 -19506.029,E2 -19506.029} C_VEL
LIN {X 0,Y 108.061,Z 752.778,A -85,B 0,C 180,E1 -19500.8,E2 -19500.8} C_VEL
LIN {X 0,Y 111.01,Z 750.259,A -85,B 0,C 180,E1 -19498.108,E2 -19498.108} C_VEL
LIN {X 0,Y 116.082,Z 753.326,A -85,B 0,C 180,E1 -19492.735,E2 -19492.735} C_VEL
LIN {X 0,Y 123.869,Z 756.242,A -85,B 0,C 180,E1 -19487.085,E2 -19487.085} C_VEL
LIN {X 0,Y 130.017,Z 757.724,A -85,B 0,C 180,E1 -19483.727,E2 -19483.727} C_VEL
LIN {X 0,Y 131.004,Z 757.786,A -85,B 0,C 180,E1 -19482.517,E2 -19482.517} C_VEL
LIN {X 0,Y 121.493,Z 753.639,A -85,B 0,C 180,E1 -19477.401,E2 -19477.401} C_VEL
LIN {X 0,Y 113.99,Z 748.54,A -85,B 0,C 180,E1 -19471.605,E2 -19471.605} C_VEL
LIN {X 0,Y 107.688,Z 741.265,A -85,B 0,C 180,E1 -19463.971,E2 -19463.971} C_VEL
LIN {X 0,Y 104.262,Z 733.341,A -85,B 0,C 180,E1 -19456.647,E2 -19456.647} C_VEL
LIN {X 0,Y 102.924,Z 724.893,A -85,B 0,C 180,E1 -19449.828,E2 -19449.828} C_VEL
LIN {X 0,Y 102.56,Z 716.064,A -85,B 0,C 180,E1 -19443.929,E2 -19443.929} C_VEL
LIN {X 0,Y 102.487,Z 712.608,A -85,B 0,C 180,E1 -19441.964,E2 -19441.964} C_VEL
LIN {X 0,Y 101.846,Z 713.028,A -85,B 0,C 180,E1 -19439.999,E2 -19439.999} C_VEL
LIN {X 0,Y 103.262,Z 711.276,A -85,B 0,C 180,E1 -19436.097,E2 -19436.097} C_VEL
LIN {X 0,Y 105.83,Z 709.126,A -85,B 0,C 180,E1 -19430.443,E2 -19430.443} C_VEL
LIN {X 0,Y 107.71,Z 707.564,A -85,B 0,C 180,E1 -19428.185,E2 -19428.185} C_VEL
LIN {X 0,Y 111.434,Z 705.217,A -85,B 0,C 180,E1 -19423.512,E2 -19423.512} C_VEL
LIN {X 0,Y 113.56,Z 703.614,A -85,B 0,C 180,E1 -19421.974,E2 -19421.974} C_VEL
LIN {X 0,Y 119.181,Z 700.163,A -85,B 0,C 180,E1 -19417.461,E2 -19417.461} C_VEL
LIN {X 0,Y 123.899,Z 696.48,A -85,B 0,C 180,E1 -19415.182,E2 -19415.182} C_VEL
LIN {X 0,Y 126.455,Z 695.004,A -85,B 0,C 180,E1 -19413.601,E2 -19413.601} C_VEL
LIN {X 0,Y 131.759,Z 691.05,A -85,B 0,C 180,E1 -19411.31,E2 -19411.31} C_VEL
LIN {X 0,Y 138.071,Z 685.153,A -85,B 0,C 180,E1 -19409.401,E2 -19409.401} C_VEL
LIN {X 0,Y 142.238,Z 681.766,A -85,B 0,C 180,E1 -19407.916,E2 -19407.916} C_VEL
LIN {X 0,Y 147.431,Z 676.597,A -85,B 0,C 180,E1 -19406.489,E2 -19406.489} C_VEL
LIN {X 0,Y 150.936,Z 672.387,A -85,B 0,C 180,E1 -19405.742,E2 -19405.742} C_VEL
LIN {X 0,Y 151.198,Z 672.747,A -85,B 0,C 180,E1 -19405.475,E2 -19405.475} C_VEL
LIN {X 0,Y 150.675,Z 675.045,A -85,B 0,C 180,E1 -19405.056,E2 -19405.056} C_VEL
LIN {X 0,Y 147.715,Z 681.37,A -85,B 0,C 180,E1 -19404.545,E2 -19404.545} C_VEL
LIN {X 0,Y 141.886,Z 690.799,A -85,B 0,C 180,E1 -19404.056,E2 -19404.056} C_VEL
LIN {X 0,Y 137.616,Z 697.473,A -85,B 0,C 180,E1 -19403.267,E2 -19403.267} C_VEL
LIN {X 0,Y 136.37,Z 699.624,A -85,B 0,C 180,E1 -19402.834,E2 -19402.834} C_VEL
LIN {X 0,Y 130.335,Z 709.644,A -85,B 0,C 180,E1 -19400.216,E2 -19400.216} C_VEL
LIN {X 0,Y 123.359,Z 719.698,A -85,B 0,C 180,E1 -19396.587,E2 -19396.587} C_VEL
LIN {X 0,Y 116.792,Z 727.842,A -85,B 0,C 180,E1 -19392.613,E2 -19392.613} C_VEL
LIN {X 0,Y 109.784,Z 735.494,A -85,B 0,C 180,E1 -19387.462,E2 -19387.462} C_VEL
LIN {X 0,Y 104.601,Z 740.7,A -85,B 0,C 180,E1 -19382.52,E2 -19382.52} C_VEL
LIN {X 0,Y 100.165,Z 744.84,A -85,B 0,C 180,E1 -19377.139,E2 -19377.139} C_VEL
LIN {X 0,Y 96.602,Z 748.023,A -85,B 0,C 180,E1 -19371.337,E2 -19371.337} C_VEL
LIN {X 0,Y 93.398,Z 750.873,A -85,B 0,C 180,E1 -19363.052,E2 -19363.052} C_VEL
LIN {X 0,Y 91.827,Z 752.287,A -85,B 0,C 180,E1 -19354.395,E2 -19354.395} C_VEL
LIN {X 0,Y 91.65,Z 752.458,A -85,B 0,C 180,E1 -19350.006,E2 -19350.006} C_VEL
LIN {X 0,Y 92.439,Z 751.712,A -85,B 0,C 180,E1 -19341.26,E2 -19341.26} C_VEL
LIN {X 0,Y 94.76,Z 749.56,A -85,B 0,C 180,E1 -19332.749,E2 -19332.749} C_VEL
LIN {X 0,Y 98.876,Z 745.909,A -85,B 0,C 180,E1 -19324.762,E2 -19324.762} C_VEL
LIN {X 0,Y 103.071,Z 742.041,A -85,B 0,C 180,E1 -19319.249,E2 -19319.249} C_VEL
LIN {X 0,Y 108.053,Z 737.151,A -85,B 0,C 180,E1 -19314.177,E2 -19314.177} C_VEL
LIN {X 0,Y 113.718,Z 731.101,A -85,B 0,C 180,E1 -19309.546,E2 -19309.546} C_VEL
LIN {X 0,Y 120.069,Z 723.678,A -85,B 0,C 180,E1 -19305.387,E2 -19305.387} C_VEL
LIN {X 0,Y 126.738,Z 714.728,A -85,B 0,C 180,E1 -19301.632,E2 -19301.632} C_VEL
LIN {X 0,Y 133.497,Z 704.256,A -85,B 0,C 180,E1 -19298.462,E2 -19298.462} C_VEL
LIN {X 0,Y 139.24,Z 693.891,A -85,B 0,C 180,E1 -19296.147,E2 -19296.147} C_VEL
LIN {X 0,Y 144.496,Z 682.53,A -85,B 0,C 180,E1 -19294.231,E2 -19294.231} C_VEL
LIN {X 0,Y 149.182,Z 669.896,A -85,B 0,C 180,E1 -19292.645,E2 -19292.645} C_VEL
LIN {X 0,Y 152.706,Z 657.137,A -85,B 0,C 180,E1 -19291.462,E2 -19291.462} C_VEL
LIN {X 0,Y 155.338,Z 643.459,A -85,B 0,C 180,E1 -19290.623,E2 -19290.623} C_VEL
LIN {X 0,Y 157.401,Z 624.196,A -85,B 0,C 180,E1 -19289.936,E2 -19289.936} C_VEL
LIN {X 0,Y 159.407,Z 601.378,A -85,B 0,C 180,E1 -19289.191,E2 -19289.191} C_VEL
LIN {X 0,Y 156.073,Z 592.711,A -85,B 0,C 180,E1 -19285.848,E2 -19285.848} C_VEL
LIN {X 0,Y 153.154,Z 585.992,A -85,B 0,C 180,E1 -19282.474,E2 -19282.474} C_VEL
LIN {X 0,Y 150.495,Z 580.496,A -85,B 0,C 180,E1 -19278.816,E2 -19278.816} C_VEL
LIN {X 0,Y 148.746,Z 577.248,A -85,B 0,C 180,E1 -19275.904,E2 -19275.904} C_VEL
LIN {X 0,Y 146.738,Z 573.286,A -85,B 0,C 180,E1 -19271.395,E2 -19271.395} C_VEL
LIN {X 0,Y 145.252,Z 570.776,A -85,B 0,C 180,E1 -19265.554,E2 -19265.554} C_VEL
LIN {X 0,Y 145.011,Z 570.165,A -85,B 0,C 180,E1 -19262.778,E2 -19262.778} C_VEL
LIN {X 0,Y 145.07,Z 570.111,A -85,B 0,C 180,E1 -19259.653,E2 -19259.653} C_VEL
LIN {X 0,Y 146.268,Z 572.747,A -85,B 0,C 180,E1 -19253.101,E2 -19253.101} C_VEL
LIN {X 0,Y 147.165,Z 574.544,A -85,B 0,C 180,E1 -19250.552,E2 -19250.552} C_VEL
LIN {X 0,Y 149.539,Z 579.292,A -85,B 0,C 180,E1 -19245.716,E2 -19245.716} C_VEL
LIN {X 0,Y 151.591,Z 583.543,A -85,B 0,C 180,E1 -19242.549,E2 -19242.549} C_VEL
LIN {X 0,Y 154.249,Z 589.352,A -85,B 0,C 180,E1 -19239.148,E2 -19239.148} C_VEL
LIN {X 0,Y 157.156,Z 596.669,A -85,B 0,C 180,E1 -19235.917,E2 -19235.917} C_VEL
LIN {X 0,Y 159.465,Z 603.098,A -85,B 0,C 180,E1 -19233.615,E2 -19233.615} C_VEL
LIN {X 0,Y 155.271,Z 645.732,A -85,B 0,C 180,E1 -19232.217,E2 -19232.217} C_VEL
LIN {X 0,Y 152.751,Z 659.482,A -85,B 0,C 180,E1 -19231.501,E2 -19231.501} C_VEL
LIN {X 0,Y 148.926,Z 673.378,A -85,B 0,C 180,E1 -19230.461,E2 -19230.461} C_VEL
LIN {X 0,Y 144.356,Z 686.039,A -85,B 0,C 180,E1 -19229.094,E2 -19229.094} C_VEL
LIN {X 0,Y 138.838,Z 698.245,A -85,B 0,C 180,E1 -19227.297,E2 -19227.297} C_VEL
LIN {X 0,Y 132.824,Z 709.278,A -85,B 0,C 180,E1 -19225.091,E2 -19225.091} C_VEL
LIN {X 0,Y 126.289,Z 719.664,A -85,B 0,C 180,E1 -19222.255,E2 -19222.255} C_VEL
LIN {X 0,Y 119.411,Z 729.346,A -85,B 0,C 180,E1 -19218.618,E2 -19218.618} C_VEL
LIN {X 0,Y 112.76,Z 737.515,A -85,B 0,C 180,E1 -19214.515,E2 -19214.515} C_VEL
LIN {X 0,Y 105.953,Z 745.271,A -85,B 0,C 180,E1 -19209.054,E2 -19209.054} C_VEL
LIN {X 0,Y 100.998,Z 750.581,A -85,B 0,C 180,E1 -19203.82,E2 -19203.82} C_VEL
LIN {X 0,Y 96.938,Z 754.845,A -85,B 0,C 180,E1 -19198.109,E2 -19198.109} C_VEL
LIN {X 0,Y 93.986,Z 758.175,A -85,B 0,C 180,E1 -19191.949,E2 -19191.949} C_VEL
LIN {X 0,Y 91.645,Z 761.226,A -85,B 0,C 180,E1 -19183.295,E2 -19183.295} C_VEL
LIN {X 0,Y 91.203,Z 762.798,A -85,B 0,C 180,E1 -19174.414,E2 -19174.414} C_VEL
LIN {X 0,Y 91.377,Z 762.992,A -85,B 0,C 180,E1 -19169.004,E2 -19169.004} C_VEL
LIN {X 0,Y 91.528,Z 762.24,A -85,B 0,C 180,E1 -19161.16,E2 -19161.16} C_VEL
LIN {X 0,Y 93.362,Z 759.983,A -85,B 0,C 180,E1 -19152.47,E2 -19152.47} C_VEL
LIN {X 0,Y 97.363,Z 756.24,A -85,B 0,C 180,E1 -19144.33,E2 -19144.33} C_VEL
LIN {X 0,Y 101.929,Z 752.368,A -85,B 0,C 180,E1 -19138.855,E2 -19138.855} C_VEL
LIN {X 0,Y 106.777,Z 748.444,A -85,B 0,C 180,E1 -19134.686,E2 -19134.686} C_VEL
LIN {X 0,Y 114.703,Z 752.639,A -85,B 0,C 180,E1 -19127.619,E2 -19127.619} C_VEL
LIN {X 0,Y 120.632,Z 754.71,A -85,B 0,C 180,E1 -19123.903,E2 -19123.903} C_VEL
LIN {X 0,Y 121.467,Z 754.799,A -85,B 0,C 180,E1 -19122.544,E2 -19122.544} C_VEL
LIN {X 0,Y 111.999,Z 749.39,A -85,B 0,C 180,E1 -19116.593,E2 -19116.593} C_VEL
LIN {X 0,Y 105.06,Z 743.245,A -85,B 0,C 180,E1 -19110.113,E2 -19110.113} C_VEL
LIN {X 0,Y 99.675,Z 734.779,A -85,B 0,C 180,E1 -19101.726,E2 -19101.726} C_VEL
LIN {X 0,Y 97.073,Z 725.39,A -85,B 0,C 180,E1 -19093.609,E2 -19093.609} C_VEL
LIN {X 0,Y 96.582,Z 720.931,A -85,B 0,C 180,E1 -19090.084,E2 -19090.084} C_VEL
LIN {X 0,Y 95.82,Z 721.041,A -85,B 0,C 180,E1 -19088.435,E2 -19088.435} C_VEL
LIN {X 0,Y 95.923,Z 719.786,A -85,B 0,C 180,E1 -19084.201,E2 -19084.201} C_VEL
LIN {X 0,Y 98.891,Z 716.026,A -85,B 0,C 180,E1 -19074.291,E2 -19074.291} C_VEL
LIN {X 0,Y 102.285,Z 713.62,A -85,B 0,C 180,E1 -19068.104,E2 -19068.104} C_VEL
LIN {X 0,Y 108.595,Z 709.806,A -85,B 0,C 180,E1 -19061.119,E2 -19061.119} C_VEL
LIN {X 0,Y 110.847,Z 708.327,A -85,B 0,C 180,E1 -19059.591,E2 -19059.591} C_VEL
LIN {X 0,Y 117.007,Z 704.929,A -85,B 0,C 180,E1 -19055.136,E2 -19055.136} C_VEL
LIN {X 0,Y 122.464,Z 701.183,A -85,B 0,C 180,E1 -19052.67,E2 -19052.67} C_VEL
LIN {X 0,Y 124.793,Z 699.924,A -85,B 0,C 180,E1 -19051.399,E2 -19051.399} C_VEL
LIN {X 0,Y 131.353,Z 695.407,A -85,B 0,C 180,E1 -19048.886,E2 -19048.886} C_VEL
LIN {X 0,Y 137.677,Z 689.996,A -85,B 0,C 180,E1 -19047.214,E2 -19047.214} C_VEL
LIN {X 0,Y 143.041,Z 685.857,A -85,B 0,C 180,E1 -19045.596,E2 -19045.596} C_VEL
LIN {X 0,Y 142.584,Z 687.483,A -85,B 0,C 180,E1 -19045.138,E2 -19045.138} C_VEL
LIN {X 0,Y 136.37,Z 699.624,A -85,B 0,C 180,E1 -19042.834,E2 -19042.834} C_VEL
LIN {X 0,Y 133.35,Z 704.26,A -85,B 0,C 180,E1 -19041.95,E2 -19041.95} C_VEL
LIN {X 0,Y 127.027,Z 711.521,A -85,B 0,C 180,E1 -19040.896,E2 -19040.896} C_VEL
LIN {X 0,Y 120.417,Z 718.326,A -85,B 0,C 180,E1 -19039.546,E2 -19039.546} C_VEL
LIN {X 0,Y 117.013,Z 722.15,A -85,B 0,C 180,E1 -19038.159,E2 -19038.159} C_VEL
LIN {X 0,Y 109.474,Z 730.659,A -85,B 0,C 180,E1 -19033.646,E2 -19033.646} C_VEL
LIN {X 0,Y 102.273,Z 737.767,A -85,B 0,C 180,E1 -19028.21,E2 -19028.21} C_VEL
LIN {X 0,Y 97.006,Z 742.609,A -85,B 0,C 180,E1 -19022.919,E2 -19022.919} C_VEL
LIN {X 0,Y 92.503,Z 746.435,A -85,B 0,C 180,E1 -19017.126,E2 -19017.126} C_VEL
LIN {X 0,Y 88.029,Z 750.042,A -85,B 0,C 180,E1 -19008.63,E2 -19008.63} C_VEL
LIN {X 0,Y 85.443,Z 752.163,A -85,B 0,C 180,E1 -18999.475,E2 -18999.475} C_VEL
LIN {X 0,Y 84.574,Z 752.866,A -85,B 0,C 180,E1 -18990.006,E2 -18990.006} C_VEL
LIN {X 0,Y 85.44,Z 752.122,A -85,B 0,C 180,E1 -18980.537,E2 -18980.537} C_VEL
LIN {X 0,Y 88.021,Z 749.969,A -85,B 0,C 180,E1 -18971.381,E2 -18971.381} C_VEL
LIN {X 0,Y 92.504,Z 746.321,A -85,B 0,C 180,E1 -18962.887,E2 -18962.887} C_VEL
LIN {X 0,Y 97.061,Z 742.452,A -85,B 0,C 180,E1 -18957.115,E2 -18957.115} C_VEL
LIN {X 0,Y 102.38,Z 737.566,A -85,B 0,C 180,E1 -18951.85,E2 -18951.85} C_VEL
LIN {X 0,Y 108.437,Z 731.519,A -85,B 0,C 180,E1 -18947.123,E2 -18947.123} C_VEL
LIN {X 0,Y 115.131,Z 724.104,A -85,B 0,C 180,E1 -18942.909,E2 -18942.909} C_VEL
LIN {X 0,Y 122.244,Z 715.037,A -85,B 0,C 180,E1 -18939.102,E2 -18939.102} C_VEL
LIN {X 0,Y 129.218,Z 704.716,A -85,B 0,C 180,E1 -18936.007,E2 -18936.007} C_VEL
LIN {X 0,Y 135.193,Z 694.378,A -85,B 0,C 180,E1 -18933.728,E2 -18933.728} C_VEL
LIN {X 0,Y 140.643,Z 683.054,A -85,B 0,C 180,E1 -18931.851,E2 -18931.851} C_VEL
LIN {X 0,Y 145.497,Z 670.479,A -85,B 0,C 180,E1 -18930.305,E2 -18930.305} C_VEL
LIN {X 0,Y 149.068,Z 658.218,A -85,B 0,C 180,E1 -18929.181,E2 -18929.181} C_VEL
LIN {X 0,Y 151.757,Z 645.252,A -85,B 0,C 180,E1 -18928.377,E2 -18928.377} C_VEL
LIN {X 0,Y 153.676,Z 629.091,A -85,B 0,C 180,E1 -18927.763,E2 -18927.763} C_VEL
LIN {X 0,Y 155.89,Z 605.672,A -85,B 0,C 180,E1 -18927.057,E2 -18927.057} C_VEL
LIN {X 0,Y 155.861,Z 604.284,A -85,B 0,C 180,E1 -18926.893,E2 -18926.893} C_VEL
LIN {X 0,Y 153.106,Z 596.69,A -85,B 0,C 180,E1 -18923.74,E2 -18923.74} C_VEL
LIN {X 0,Y 150.659,Z 590.833,A -85,B 0,C 180,E1 -18920.533,E2 -18920.533} C_VEL
LIN {X 0,Y 148.825,Z 586.765,A -85,B 0,C 180,E1 -18917.698,E2 -18917.698} C_VEL
LIN {X 0,Y 147.193,Z 583.565,A -85,B 0,C 180,E1 -18914.695,E2 -18914.695} C_VEL
LIN {X 0,Y 145.511,Z 579.971,A -85,B 0,C 180,E1 -18910.435,E2 -18910.435} C_VEL
LIN {X 0,Y 144.295,Z 577.689,A -85,B 0,C 180,E1 -18904.89,E2 -18904.89} C_VEL
LIN {X 0,Y 144.185,Z 577.1,A -85,B 0,C 180,E1 -18900,E2 -18900} C_VEL
LIN {X 0,Y 145.281,Z 579.769,A -85,B 0,C 180,E1 -18893.403,E2 -18893.403} C_VEL
LIN {X 0,Y 146.059,Z 581.538,A -85,B 0,C 180,E1 -18891.003,E2 -18891.003} C_VEL
LIN {X 0,Y 148.093,Z 585.944,A -85,B 0,C 180,E1 -18886.536,E2 -18886.536} C_VEL
LIN {X 0,Y 149.967,Z 590.146,A -85,B 0,C 180,E1 -18883.407,E2 -18883.407} C_VEL
LIN {X 0,Y 152.4,Z 596.015,A -85,B 0,C 180,E1 -18880.029,E2 -18880.029} C_VEL
LIN {X 0,Y 155.291,Z 603.971,A -85,B 0,C 180,E1 -18876.584,E2 -18876.584} C_VEL
LIN {X 0,Y 156.002,Z 606.177,A -85,B 0,C 180,E1 -18875.794,E2 -18875.794} C_VEL
LIN {X 0,Y 151.828,Z 646.291,A -85,B 0,C 180,E1 -18874.527,E2 -18874.527} C_VEL
LIN {X 0,Y 149.048,Z 660.513,A -85,B 0,C 180,E1 -18873.793,E2 -18873.793} C_VEL
LIN {X 0,Y 145.186,Z 673.883,A -85,B 0,C 180,E1 -18872.799,E2 -18872.799} C_VEL
LIN {X 0,Y 140.111,Z 687.213,A -85,B 0,C 180,E1 -18871.37,E2 -18871.37} C_VEL
LIN {X 0,Y 134.43,Z 699.061,A -85,B 0,C 180,E1 -18869.604,E2 -18869.604} C_VEL
LIN {X 0,Y 127.515,Z 710.971,A -85,B 0,C 180,E1 -18867.185,E2 -18867.185} C_VEL
LIN {X 0,Y 120.98,Z 720.736,A -85,B 0,C 180,E1 -18864.41,E2 -18864.41} C_VEL
LIN {X 0,Y 113.62,Z 730.418,A -85,B 0,C 180,E1 -18860.633,E2 -18860.633} C_VEL
LIN {X 0,Y 106.642,Z 738.332,A -85,B 0,C 180,E1 -18856.455,E2 -18856.455} C_VEL
LIN {X 0,Y 100.47,Z 744.847,A -85,B 0,C 180,E1 -18851.639,E2 -18851.639} C_VEL
LIN {X 0,Y 95.137,Z 750.163,A -85,B 0,C 180,E1 -18846.219,E2 -18846.219} C_VEL
LIN {X 0,Y 90.675,Z 754.429,A -85,B 0,C 180,E1 -18840.245,E2 -18840.245} C_VEL
LIN {X 0,Y 87.39,Z 757.761,A -85,B 0,C 180,E1 -18833.703,E2 -18833.703} C_VEL
LIN {X 0,Y 84.699,Z 760.812,A -85,B 0,C 180,E1 -18824.407,E2 -18824.407} C_VEL
LIN {X 0,Y 84.089,Z 762.386,A -85,B 0,C 180,E1 -18814.788,E2 -18814.788} C_VEL
LIN {X 0,Y 84.335,Z 762.613,A -85,B 0,C 180,E1 -18809.994,E2 -18809.994} C_VEL
LIN {X 0,Y 84.221,Z 762.41,A -85,B 0,C 180,E1 -18805.207,E2 -18805.207} C_VEL
LIN {X 0,Y 85.241,Z 760.881,A -85,B 0,C 180,E1 -18795.673,E2 -18795.673} C_VEL
LIN {X 0,Y 88.539,Z 757.893,A -85,B 0,C 180,E1 -18786.61,E2 -18786.61} C_VEL
LIN {X 0,Y 92.562,Z 754.643,A -85,B 0,C 180,E1 -18780.421,E2 -18780.421} C_VEL
LIN {X 0,Y 97.828,Z 750.472,A -85,B 0,C 180,E1 -18774.914,E2 -18774.914} C_VEL
LIN {X 0,Y 102.894,Z 746.509,A -85,B 0,C 180,E1 -18771.125,E2 -18771.125} C_VEL
LIN {X 0,Y 113.165,Z 751.445,A -85,B 0,C 180,E1 -18763.089,E2 -18763.089} C_VEL
LIN {X 0,Y 104.594,Z 745.737,A -85,B 0,C 180,E1 -18757.209,E2 -18757.209} C_VEL
LIN {X 0,Y 97.199,Z 737.904,A -85,B 0,C 180,E1 -18749.252,E2 -18749.252} C_VEL
LIN {X 0,Y 92.692,Z 729.334,A -85,B 0,C 180,E1 -18740.963,E2 -18740.963} C_VEL
LIN {X 0,Y 90.971,Z 729.063,A -85,B 0,C 180,E1 -18738,E2 -18738} C_VEL
LIN {X 0,Y 90.306,Z 727.596,A -85,B 0,C 180,E1 -18733.501,E2 -18733.501} C_VEL
LIN {X 0,Y 90.586,Z 725.753,A -85,B 0,C 180,E1 -18728.926,E2 -18728.926} C_VEL
LIN {X 0,Y 90.574,Z 724.641,A -85,B 0,C 180,E1 -18724.45,E2 -18724.45} C_VEL
LIN {X 0,Y 97.182,Z 718.811,A -85,B 0,C 180,E1 -18707.469,E2 -18707.469} C_VEL
LIN {X 0,Y 105.688,Z 714.249,A -85,B 0,C 180,E1 -18698.598,E2 -18698.598} C_VEL
LIN {X 0,Y 108.118,Z 712.858,A -85,B 0,C 180,E1 -18697.044,E2 -18697.044} C_VEL
LIN {X 0,Y 114.852,Z 709.489,A -85,B 0,C 180,E1 -18692.681,E2 -18692.681} C_VEL
LIN {X 0,Y 120.611,Z 705.937,A -85,B 0,C 180,E1 -18690.308,E2 -18690.308} C_VEL
LIN {X 0,Y 123.12,Z 704.674,A -85,B 0,C 180,E1 -18689.086,E2 -18689.086} C_VEL
LIN {X 0,Y 129.029,Z 701.039,A -85,B 0,C 180,E1 -18686.996,E2 -18686.996} C_VEL
LIN {X 0,Y 132.419,Z 698.608,A -85,B 0,C 180,E1 -18686.055,E2 -18686.055} C_VEL
LIN {X 0,Y 132.418,Z 699.732,A -85,B 0,C 180,E1 -18685.358,E2 -18685.358} C_VEL
LIN {X 0,Y 125.932,Z 710.089,A -85,B 0,C 180,E1 -18682.686,E2 -18682.686} C_VEL
LIN {X 0,Y 119.808,Z 718.601,A -85,B 0,C 180,E1 -18679.699,E2 -18679.699} C_VEL
LIN {X 0,Y 117.013,Z 722.15,A -85,B 0,C 180,E1 -18678.159,E2 -18678.159} C_VEL
LIN {X 0,Y 113.528,Z 725.824,A -85,B 0,C 180,E1 -18676.646,E2 -18676.646} C_VEL
LIN {X 0,Y 106.372,Z 731.439,A -85,B 0,C 180,E1 -18674.566,E2 -18674.566} C_VEL
LIN {X 0,Y 99.125,Z 736.519,A -85,B 0,C 180,E1 -18672.028,E2 -18672.028} C_VEL
LIN {X 0,Y 95.619,Z 739.239,A -85,B 0,C 180,E1 -18669.752,E2 -18669.752} C_VEL
LIN {X 0,Y 89.428,Z 744.413,A -85,B 0,C 180,E1 -18663.382,E2 -18663.382} C_VEL
LIN {X 0,Y 86.25,Z 746.844,A -85,B 0,C 180,E1 -18659.275,E2 -18659.275} C_VEL
LIN {X 0,Y 81.342,Z 750.451,A -85,B 0,C 180,E1 -18650.225,E2 -18650.225} C_VEL
LIN {X 0,Y 78.463,Z 752.571,A -85,B 0,C 180,E1 -18640.326,E2 -18640.326} C_VEL
LIN {X 0,Y 77.487,Z 753.275,A -85,B 0,C 180,E1 -18630.007,E2 -18630.007} C_VEL
LIN {X 0,Y 78.46,Z 752.531,A -85,B 0,C 180,E1 -18619.687,E2 -18619.687} C_VEL
LIN {X 0,Y 81.333,Z 750.379,A -85,B 0,C 180,E1 -18609.786,E2 -18609.786} C_VEL
LIN {X 0,Y 86.25,Z 746.732,A -85,B 0,C 180,E1 -18600.739,E2 -18600.739} C_VEL
LIN {X 0,Y 91.187,Z 742.864,A -85,B 0,C 180,E1 -18594.694,E2 -18594.694} C_VEL
LIN {X 0,Y 96.895,Z 737.982,A -85,B 0,C 180,E1 -18589.256,E2 -18589.256} C_VEL
LIN {X 0,Y 103.372,Z 731.937,A -85,B 0,C 180,E1 -18584.457,E2 -18584.457} C_VEL
LIN {X 0,Y 110.432,Z 724.53,A -85,B 0,C 180,E1 -18580.217,E2 -18580.217} C_VEL
LIN {X 0,Y 117.905,Z 715.477,A -85,B 0,C 180,E1 -18576.43,E2 -18576.43} C_VEL
LIN {X 0,Y 125.199,Z 705.177,A -85,B 0,C 180,E1 -18573.392,E2 -18573.392} C_VEL
LIN {X 0,Y 131.403,Z 694.864,A -85,B 0,C 180,E1 -18571.166,E2 -18571.166} C_VEL
LIN {X 0,Y 137.044,Z 683.579,A -85,B 0,C 180,E1 -18569.34,E2 -18569.34} C_VEL
LIN {X 0,Y 142.069,Z 671.062,A -85,B 0,C 180,E1 -18567.848,E2 -18567.848} C_VEL
LIN {X 0,Y 145.98,Z 658.026,A -85,B 0,C 180,E1 -18566.685,E2 -18566.685} C_VEL
LIN {X 0,Y 148.78,Z 644.589,A -85,B 0,C 180,E1 -18565.894,E2 -18565.894} C_VEL
LIN {X 0,Y 150.883,Z 626.916,A -85,B 0,C 180,E1 -18565.286,E2 -18565.286} C_VEL
LIN {X 0,Y 152.761,Z 607.872,A -85,B 0,C 180,E1 -18564.739,E2 -18564.739} C_VEL
LIN {X 0,Y 150.458,Z 601.122,A -85,B 0,C 180,E1 -18561.734,E2 -18561.734} C_VEL
LIN {X 0,Y 148.378,Z 595.831,A -85,B 0,C 180,E1 -18558.605,E2 -18558.605} C_VEL
LIN {X 0,Y 146.92,Z 592.436,A -85,B 0,C 180,E1 -18556.011,E2 -18556.011} C_VEL
LIN {X 0,Y 145.696,Z 589.812,A -85,B 0,C 180,E1 -18553.424,E2 -18553.424} C_VEL
LIN {X 0,Y 144.432,Z 586.815,A -85,B 0,C 180,E1 -18549.806,E2 -18549.806} C_VEL
LIN {X 0,Y 143.359,Z 584.601,A -85,B 0,C 180,E1 -18544.218,E2 -18544.218} C_VEL
LIN {X 0,Y 143.309,Z 584.234,A -85,B 0,C 180,E1 -18540,E2 -18540} C_VEL
LIN {X 0,Y 144.199,Z 586.592,A -85,B 0,C 180,E1 -18534.056,E2 -18534.056} C_VEL
LIN {X 0,Y 144.903,Z 588.406,A -85,B 0,C 180,E1 -18531.634,E2 -18531.634} C_VEL
LIN {X 0,Y 146.6,Z 592.366,A -85,B 0,C 180,E1 -18527.542,E2 -18527.542} C_VEL
LIN {X 0,Y 148.322,Z 596.664,A -85,B 0,C 180,E1 -18524.366,E2 -18524.366} C_VEL
LIN {X 0,Y 150.593,Z 602.67,A -85,B 0,C 180,E1 -18520.933,E2 -18520.933} C_VEL
LIN {X 0,Y 152.73,Z 609.106,A -85,B 0,C 180,E1 -18518.125,E2 -18518.125} C_VEL
LIN {X 0,Y 148.781,Z 646.008,A -85,B 0,C 180,E1 -18516.976,E2 -18516.976} C_VEL
LIN {X 0,Y 146.017,Z 659.889,A -85,B 0,C 180,E1 -18516.286,E2 -18516.286} C_VEL
LIN {X 0,Y 142.084,Z 673.258,A -85,B 0,C 180,E1 -18515.343,E2 -18515.343} C_VEL
LIN {X 0,Y 136.851,Z 686.68,A -85,B 0,C 180,E1 -18513.98,E2 -18513.98} C_VEL
LIN {X 0,Y 130.956,Z 698.568,A -85,B 0,C 180,E1 -18512.304,E2 -18512.304} C_VEL
LIN {X 0,Y 123.785,Z 710.503,A -85,B 0,C 180,E1 -18509.969,E2 -18509.969} C_VEL
LIN {X 0,Y 116.812,Z 720.466,A -85,B 0,C 180,E1 -18507.216,E2 -18507.216} C_VEL
LIN {X 0,Y 109.217,Z 729.981,A -85,B 0,C 180,E1 -18503.54,E2 -18503.54} C_VEL
LIN {X 0,Y 101.846,Z 737.905,A -85,B 0,C 180,E1 -18499.374,E2 -18499.374} C_VEL
LIN {X 0,Y 95.229,Z 744.424,A -85,B 0,C 180,E1 -18494.508,E2 -18494.508} C_VEL
LIN {X 0,Y 89.451,Z 749.744,A -85,B 0,C 180,E1 -18488.935,E2 -18488.935} C_VEL
LIN {X 0,Y 84.542,Z 754.011,A -85,B 0,C 180,E1 -18482.699,E2 -18482.699} C_VEL
LIN {X 0,Y 80.862,Z 757.345,A -85,B 0,C 180,E1 -18475.75,E2 -18475.75} C_VEL
LIN {X 0,Y 77.801,Z 760.4,A -85,B 0,C 180,E1 -18465.717,E2 -18465.717} C_VEL
LIN {X 0,Y 76.988,Z 761.975,A -85,B 0,C 180,E1 -18455.231,E2 -18455.231} C_VEL
LIN {X 0,Y 77.228,Z 762.203,A -85,B 0,C 180,E1 -18449.993,E2 -18449.993} C_VEL
LIN {X 0,Y 77.149,Z 762.001,A -85,B 0,C 180,E1 -18444.767,E2 -18444.767} C_VEL
LIN {X 0,Y 78.383,Z 760.472,A -85,B 0,C 180,E1 -18434.389,E2 -18434.389} C_VEL
LIN {X 0,Y 82.049,Z 757.482,A -85,B 0,C 180,E1 -18424.635,E2 -18424.635} C_VEL
LIN {X 0,Y 86.474,Z 754.233,A -85,B 0,C 180,E1 -18418.104,E2 -18418.104} C_VEL
LIN {X 0,Y 92.133,Z 750.061,A -85,B 0,C 180,E1 -18412.386,E2 -18412.386} C_VEL
LIN {X 0,Y 99.312,Z 744.624,A -85,B 0,C 180,E1 -18407.406,E2 -18407.406} C_VEL
LIN {X 0,Y 99.642,Z 744.435,A -85,B 0,C 180,E1 -18407.238,E2 -18407.238} C_VEL
LIN {X 0,Y 101.098,Z 745.271,A -85,B 0,C 180,E1 -18405.953,E2 -18405.953} C_VEL
LIN {X 0,Y 103.688,Z 746.441,A -85,B 0,C 180,E1 -18402.671,E2 -18402.671} C_VEL
LIN {X 0,Y 95.631,Z 739.717,A -85,B 0,C 180,E1 -18396.009,E2 -18396.009} C_VEL
LIN {X 0,Y 92.887,Z 736.706,A -85,B 0,C 180,E1 -18392.943,E2 -18392.943} C_VEL
LIN {X 0,Y 92.083,Z 736.706,A -85,B 0,C 180,E1 -18392.293,E2 -18392.293} C_VEL
LIN {X 0,Y 88.958,Z 735.946,A -85,B 0,C 180,E1 -18388.295,E2 -18388.295} C_VEL
LIN {X 0,Y 87.234,Z 734.467,A -85,B 0,C 180,E1 -18383.754,E2 -18383.754} C_VEL
LIN {X 0,Y 84.683,Z 732.104,A -85,B 0,C 180,E1 -18374.416,E2 -18374.416} C_VEL
LIN {X 0,Y 84.958,Z 729.673,A -85,B 0,C 180,E1 -18366.888,E2 -18366.888} C_VEL
LIN {X 0,Y 91.858,Z 723.702,A -85,B 0,C 180,E1 -18346.73,E2 -18346.73} C_VEL
LIN {X 0,Y 98.716,Z 720.375,A -85,B 0,C 180,E1 -18339.146,E2 -18339.146} C_VEL
LIN {X 0,Y 102.934,Z 718.421,A -85,B 0,C 180,E1 -18335.816,E2 -18335.816} C_VEL
LIN {X 0,Y 107.72,Z 716.192,A -85,B 0,C 180,E1 -18332.825,E2 -18332.825} C_VEL
LIN {X 0,Y 112.73,Z 713.858,A -85,B 0,C 180,E1 -18330.082,E2 -18330.082} C_VEL
LIN {X 0,Y 118.775,Z 710.5,A -85,B 0,C 180,E1 -18327.822,E2 -18327.822} C_VEL
LIN {X 0,Y 122.46,Z 708.692,A -85,B 0,C 180,E1 -18326.315,E2 -18326.315} C_VEL
LIN {X 0,Y 122.381,Z 709.63,A -85,B 0,C 180,E1 -18325.603,E2 -18325.603} C_VEL
LIN {X 0,Y 115.354,Z 719.034,A -85,B 0,C 180,E1 -18322.383,E2 -18322.383} C_VEL
LIN {X 0,Y 108.008,Z 727.463,A -85,B 0,C 180,E1 -18318.45,E2 -18318.45} C_VEL
LIN {X 0,Y 101.071,Z 734.339,A -85,B 0,C 180,E1 -18314.062,E2 -18314.062} C_VEL
LIN {X 0,Y 95.619,Z 739.239,A -85,B 0,C 180,E1 -18309.752,E2 -18309.752} C_VEL
LIN {X 0,Y 92.23,Z 741.78,A -85,B 0,C 180,E1 -18307.241,E2 -18307.241} C_VEL
LIN {X 0,Y 85.365,Z 745.49,A -85,B 0,C 180,E1 -18303.284,E2 -18303.284} C_VEL
LIN {X 0,Y 79.954,Z 747.978,A -85,B 0,C 180,E1 -18299.609,E2 -18299.609} C_VEL
LIN {X 0,Y 76.747,Z 749.574,A -85,B 0,C 180,E1 -18296.146,E2 -18296.146} C_VEL
LIN {X 0,Y 75.972,Z 749.994,A -85,B 0,C 180,E1 -18294.826,E2 -18294.826} C_VEL
LIN {X 0,Y 72.844,Z 752.099,A -85,B 0,C 180,E1 -18286.832,E2 -18286.832} C_VEL
LIN {X 0,Y 70.672,Z 753.512,A -85,B 0,C 180,E1 -18275.715,E2 -18275.715} C_VEL
LIN {X 0,Y 70.41,Z 753.684,A -85,B 0,C 180,E1 -18270.007,E2 -18270.007} C_VEL
LIN {X 0,Y 71.515,Z 752.939,A -85,B 0,C 180,E1 -18258.673,E2 -18258.673} C_VEL
LIN {X 0,Y 74.711,Z 750.789,A -85,B 0,C 180,E1 -18247.905,E2 -18247.905} C_VEL
LIN {X 0,Y 80.142,Z 747.142,A -85,B 0,C 180,E1 -18238.261,E2 -18238.261} C_VEL
LIN {X 0,Y 85.504,Z 743.276,A -85,B 0,C 180,E1 -18231.95,E2 -18231.95} C_VEL
LIN {X 0,Y 91.634,Z 738.397,A -85,B 0,C 180,E1 -18226.357,E2 -18226.357} C_VEL
LIN {X 0,Y 98.551,Z 732.356,A -85,B 0,C 180,E1 -18221.523,E2 -18221.523} C_VEL
LIN {X 0,Y 106,Z 724.957,A -85,B 0,C 180,E1 -18217.295,E2 -18217.295} C_VEL
LIN {X 0,Y 113.849,Z 715.916,A -85,B 0,C 180,E1 -18213.566,E2 -18213.566} C_VEL
LIN {X 0,Y 121.453,Z 705.639,A -85,B 0,C 180,E1 -18210.608,E2 -18210.608} C_VEL
LIN {X 0,Y 127.893,Z 695.351,A -85,B 0,C 180,E1 -18208.459,E2 -18208.459} C_VEL
LIN {X 0,Y 133.722,Z 684.104,A -85,B 0,C 180,E1 -18206.698,E2 -18206.698} C_VEL
LIN {X 0,Y 138.913,Z 671.644,A -85,B 0,C 180,E1 -18205.275,E2 -18205.275} C_VEL
LIN {X 0,Y 142.837,Z 659.15,A -85,B 0,C 180,E1 -18204.189,E2 -18204.189} C_VEL
LIN {X 0,Y 145.755,Z 646.123,A -85,B 0,C 180,E1 -18203.427,E2 -18203.427} C_VEL
LIN {X 0,Y 147.802,Z 630.387,A -85,B 0,C 180,E1 -18202.871,E2 -18202.871} C_VEL
LIN {X 0,Y 149.768,Z 611.04,A -85,B 0,C 180,E1 -18202.333,E2 -18202.333} C_VEL
LIN {X 0,Y 147.724,Z 604.877,A -85,B 0,C 180,E1 -18199.225,E2 -18199.225} C_VEL
LIN {X 0,Y 145.693,Z 599.406,A -85,B 0,C 180,E1 -18195.478,E2 -18195.478} C_VEL
LIN {X 0,Y 144.459,Z 596.536,A -85,B 0,C 180,E1 -18192.647,E2 -18192.647} C_VEL
LIN {X 0,Y 143.281,Z 593.459,A -85,B 0,C 180,E1 -18188.818,E2 -18188.818} C_VEL
LIN {X 0,Y 142.443,Z 591.515,A -85,B 0,C 180,E1 -18183.536,E2 -18183.536} C_VEL
LIN {X 0,Y 142.444,Z 591.482,A -85,B 0,C 180,E1 -18179.647,E2 -18179.647} C_VEL
LIN {X 0,Y 143.135,Z 593.416,A -85,B 0,C 180,E1 -18174.718,E2 -18174.718} C_VEL
LIN {X 0,Y 143.765,Z 595.263,A -85,B 0,C 180,E1 -18172.274,E2 -18172.274} C_VEL
LIN {X 0,Y 145.145,Z 598.841,A -85,B 0,C 180,E1 -18168.567,E2 -18168.567} C_VEL
LIN {X 0,Y 146.555,Z 602.684,A -85,B 0,C 180,E1 -18165.657,E2 -18165.657} C_VEL
LIN {X 0,Y 148.376,Z 607.974,A -85,B 0,C 180,E1 -18162.547,E2 -18162.547} C_VEL
LIN {X 0,Y 149.729,Z 612.421,A -85,B 0,C 180,E1 -18160.495,E2 -18160.495} C_VEL
LIN {X 0,Y 146.002,Z 645.809,A -85,B 0,C 180,E1 -18159.52,E2 -18159.52} C_VEL
LIN {X 0,Y 143.151,Z 659.714,A -85,B 0,C 180,E1 -18158.865,E2 -18158.865} C_VEL
LIN {X 0,Y 139.275,Z 672.633,A -85,B 0,C 180,E1 -18157.995,E2 -18157.995} C_VEL
LIN {X 0,Y 134.642,Z 684.377,A -85,B 0,C 180,E1 -18156.912,E2 -18156.912} C_VEL
LIN {X 0,Y 128.553,Z 696.741,A -85,B 0,C 180,E1 -18155.342,E2 -18155.342} C_VEL
LIN {X 0,Y 121.85,Z 707.883,A -85,B 0,C 180,E1 -18153.37,E2 -18153.37} C_VEL
LIN {X 0,Y 114.654,Z 718.036,A -85,B 0,C 180,E1 -18150.856,E2 -18150.856} C_VEL
LIN {X 0,Y 107.799,Z 726.531,A -85,B 0,C 180,E1 -18147.935,E2 -18147.935} C_VEL
LIN {X 0,Y 99.901,Z 734.983,A -85,B 0,C 180,E1 -18143.991,E2 -18143.991} C_VEL
LIN {X 0,Y 92.548,Z 741.946,A -85,B 0,C 180,E1 -18139.401,E2 -18139.401} C_VEL
LIN {X 0,Y 86,Z 747.671,A -85,B 0,C 180,E1 -18133.989,E2 -18133.989} C_VEL
LIN {X 0,Y 80.227,Z 752.304,A -85,B 0,C 180,E1 -18127.814,E2 -18127.814} C_VEL
LIN {X 0,Y 74.466,Z 756.93,A -85,B 0,C 180,E1 -18118.149,E2 -18118.149} C_VEL
LIN {X 0,Y 70.922,Z 759.985,A -85,B 0,C 180,E1 -18107.287,E2 -18107.287} C_VEL
LIN {X 0,Y 69.889,Z 761.563,A -85,B 0,C 180,E1 -18095.764,E2 -18095.764} C_VEL
LIN {X 0,Y 70.129,Z 761.794,A -85,B 0,C 180,E1 -18089.993,E2 -18089.993} C_VEL
LIN {X 0,Y 70.074,Z 761.591,A -85,B 0,C 180,E1 -18084.236,E2 -18084.236} C_VEL
LIN {X 0,Y 71.547,Z 760.061,A -85,B 0,C 180,E1 -18072.854,E2 -18072.854} C_VEL
LIN {X 0,Y 75.674,Z 757.071,A -85,B 0,C 180,E1 -18062.324,E2 -18062.324} C_VEL
LIN {X 0,Y 80.526,Z 753.823,A -85,B 0,C 180,E1 -18055.431,E2 -18055.431} C_VEL
LIN {X 0,Y 86.642,Z 749.65,A -85,B 0,C 180,E1 -18049.532,E2 -18049.532} C_VEL
LIN {X 0,Y 94.869,Z 743.648,A -85,B 0,C 180,E1 -18044.054,E2 -18044.054} C_VEL
LIN {X 0,Y 94.038,Z 742.678,A -85,B 0,C 180,E1 -18042.269,E2 -18042.269} C_VEL
LIN {X 0,Y 90.093,Z 741.801,A -85,B 0,C 180,E1 -18038.613,E2 -18038.613} C_VEL
LIN {X 0,Y 87.098,Z 740.534,A -85,B 0,C 180,E1 -18034.39,E2 -18034.39} C_VEL
LIN {X 0,Y 83.74,Z 739.829,A -85,B 0,C 180,E1 -18030.235,E2 -18030.235} C_VEL
LIN {X 0,Y 78.9,Z 736.245,A -85,B 0,C 180,E1 -18015.498,E2 -18015.498} C_VEL
LIN {X 0,Y 79.205,Z 733.47,A -85,B 0,C 180,E1 -18005.09,E2 -18005.09} C_VEL
LIN {X 0,Y 89.605,Z 726.819,A -85,B 0,C 180,E1 -17981.715,E2 -17981.715} C_VEL
LIN {X 0,Y 100.199,Z 722.413,A -85,B 0,C 180,E1 -17972.876,E2 -17972.876} C_VEL
LIN {X 0,Y 107.873,Z 719.262,A -85,B 0,C 180,E1 -17968.586,E2 -17968.586} C_VEL
LIN {X 0,Y 112.425,Z 717.135,A -85,B 0,C 180,E1 -17966.739,E2 -17966.739} C_VEL
LIN {X 0,Y 112.303,Z 718.088,A -85,B 0,C 180,E1 -17965.795,E2 -17965.795} C_VEL
LIN {X 0,Y 104.712,Z 726.574,A -85,B 0,C 180,E1 -17962.065,E2 -17962.065} C_VEL
LIN {X 0,Y 97.298,Z 733.691,A -85,B 0,C 180,E1 -17957.77,E2 -17957.77} C_VEL
LIN {X 0,Y 89.453,Z 740.35,A -85,B 0,C 180,E1 -17951.906,E2 -17951.906} C_VEL
LIN {X 0,Y 83.599,Z 744.824,A -85,B 0,C 180,E1 -17946.056,E2 -17946.056} C_VEL
LIN {X 0,Y 80.142,Z 747.252,A -85,B 0,C 180,E1 -17941.754,E2 -17941.754} C_VEL
LIN {X 0,Y 75.972,Z 749.994,A -85,B 0,C 180,E1 -17934.826,E2 -17934.826} C_VEL
LIN {X 0,Y 73.489,Z 751.303,A -85,B 0,C 180,E1 -17930.825,E2 -17930.825} C_VEL
LIN {X 0,Y 68.418,Z 752.907,A -85,B 0,C 180,E1 -17924.056,E2 -17924.056} C_VEL
LIN {X 0,Y 64.887,Z 753.73,A -85,B 0,C 180,E1 -17917.942,E2 -17917.942} C_VEL
LIN {X 0,Y 63.455,Z 754.031,A -85,B 0,C 180,E1 -17912.799,E2 -17912.799} C_VEL
LIN {X 0,Y 63.338,Z 754.064,A -85,B 0,C 180,E1 -17911.013,E2 -17911.013} C_VEL
LIN {X 0,Y 63.641,Z 753.896,A -85,B 0,C 180,E1 -17903.668,E2 -17903.668} C_VEL
LIN {X 0,Y 66.096,Z 752.453,A -85,B 0,C 180,E1 -17891.407,E2 -17891.407} C_VEL
LIN {X 0,Y 70.929,Z 749.57,A -85,B 0,C 180,E1 -17880.311,E2 -17880.311} C_VEL
LIN {X 0,Y 76.025,Z 746.352,A -85,B 0,C 180,E1 -17873.076,E2 -17873.076} C_VEL
LIN {X 0,Y 82.185,Z 742.175,A -85,B 0,C 180,E1 -17866.843,E2 -17866.843} C_VEL
LIN {X 0,Y 89.029,Z 736.943,A -85,B 0,C 180,E1 -17861.425,E2 -17861.425} C_VEL
LIN {X 0,Y 97.91,Z 729.262,A -85,B 0,C 180,E1 -17856.155,E2 -17856.155} C_VEL
LIN {X 0,Y 105.216,Z 721.899,A -85,B 0,C 180,E1 -17852.609,E2 -17852.609} C_VEL
LIN {X 0,Y 112.92,Z 712.852,A -85,B 0,C 180,E1 -17849.395,E2 -17849.395} C_VEL
LIN {X 0,Y 120.188,Z 702.922,A -85,B 0,C 180,E1 -17846.917,E2 -17846.917} C_VEL
LIN {X 0,Y 126.964,Z 691.948,A -85,B 0,C 180,E1 -17844.995,E2 -17844.995} C_VEL
LIN {X 0,Y 132.246,Z 681.45,A -85,B 0,C 180,E1 -17843.56,E2 -17843.56} C_VEL
LIN {X 0,Y 136.822,Z 670.207,A -85,B 0,C 180,E1 -17842.406,E2 -17842.406} C_VEL
LIN {X 0,Y 140.9,Z 656.738,A -85,B 0,C 180,E1 -17841.342,E2 -17841.342} C_VEL
LIN {X 0,Y 143.807,Z 642.849,A -85,B 0,C 180,E1 -17840.656,E2 -17840.656} C_VEL
LIN {X 0,Y 146.959,Z 615.301,A -85,B 0,C 180,E1 -17839.89,E2 -17839.89} C_VEL
LIN {X 0,Y 146.966,Z 614.231,A -85,B 0,C 180,E1 -17839.739,E2 -17839.739} C_VEL
LIN {X 0,Y 145.25,Z 608.785,A -85,B 0,C 180,E1 -17836.606,E2 -17836.606} C_VEL
LIN {X 0,Y 144.022,Z 605.257,A -85,B 0,C 180,E1 -17833.901,E2 -17833.901} C_VEL
LIN {X 0,Y 142.774,Z 601.943,A -85,B 0,C 180,E1 -17830.356,E2 -17830.356} C_VEL
LIN {X 0,Y 142.248,Z 600.32,A -85,B 0,C 180,E1 -17828.212,E2 -17828.212} C_VEL
LIN {X 0,Y 141.58,Z 598.597,A -85,B 0,C 180,E1 -17823.558,E2 -17823.558} C_VEL
LIN {X 0,Y 141.558,Z 598.595,A -85,B 0,C 180,E1 -17819.645,E2 -17819.645} C_VEL
LIN {X 0,Y 142.2,Z 600.536,A -85,B 0,C 180,E1 -17814.861,E2 -17814.861} C_VEL
LIN {X 0,Y 143.68,Z 605.046,A -85,B 0,C 180,E1 -17809.788,E2 -17809.788} C_VEL
LIN {X 0,Y 145.045,Z 609.231,A -85,B 0,C 180,E1 -17806.605,E2 -17806.605} C_VEL
LIN {X 0,Y 146.693,Z 614.697,A -85,B 0,C 180,E1 -17803.474,E2 -17803.474} C_VEL
LIN {X 0,Y 146.955,Z 615.737,A -85,B 0,C 180,E1 -17803.004,E2 -17803.004} C_VEL
LIN {X 0,Y 143.462,Z 645.998,A -85,B 0,C 180,E1 -17802.133,E2 -17802.133} C_VEL
LIN {X 0,Y 140.533,Z 659.722,A -85,B 0,C 180,E1 -17801.54,E2 -17801.54} C_VEL
LIN {X 0,Y 136.364,Z 673.136,A -85,B 0,C 180,E1 -17800.686,E2 -17800.686} C_VEL
LIN {X 0,Y 131.224,Z 685.594,A -85,B 0,C 180,E1 -17799.582,E2 -17799.582} C_VEL
LIN {X 0,Y 124.971,Z 697.587,A -85,B 0,C 180,E1 -17798.099,E2 -17798.099} C_VEL
LIN {X 0,Y 118.065,Z 708.497,A -85,B 0,C 180,E1 -17796.225,E2 -17796.225} C_VEL
LIN {X 0,Y 109.882,Z 719.389,A -85,B 0,C 180,E1 -17793.552,E2 -17793.552} C_VEL
LIN {X 0,Y 102.757,Z 727.6,A -85,B 0,C 180,E1 -17790.684,E2 -17790.684} C_VEL
LIN {X 0,Y 94.529,Z 735.806,A -85,B 0,C 180,E1 -17786.752,E2 -17786.752} C_VEL
LIN {X 0,Y 86.82,Z 742.551,A -85,B 0,C 180,E1 -17782.105,E2 -17782.105} C_VEL
LIN {X 0,Y 78.805,Z 748.904,A -85,B 0,C 180,E1 -17775.507,E2 -17775.507} C_VEL
LIN {X 0,Y 72.86,Z 753.176,A -85,B 0,C 180,E1 -17768.818,E2 -17768.818} C_VEL
LIN {X 0,Y 68.23,Z 756.515,A -85,B 0,C 180,E1 -17760.99,E2 -17760.99} C_VEL
LIN {X 0,Y 64.115,Z 759.571,A -85,B 0,C 180,E1 -17749.19,E2 -17749.19} C_VEL
LIN {X 0,Y 62.793,Z 761.151,A -85,B 0,C 180,E1 -17736.418,E2 -17736.418} C_VEL
LIN {X 0,Y 63.015,Z 761.383,A -85,B 0,C 180,E1 -17729.992,E2 -17729.992} C_VEL
LIN {X 0,Y 63.006,Z 761.181,A -85,B 0,C 180,E1 -17723.587,E2 -17723.587} C_VEL
LIN {X 0,Y 64.783,Z 759.651,A -85,B 0,C 180,E1 -17710.998,E2 -17710.998} C_VEL
LIN {X 0,Y 69.447,Z 756.661,A -85,B 0,C 180,E1 -17699.594,E2 -17699.594} C_VEL
LIN {X 0,Y 74.786,Z 753.412,A -85,B 0,C 180,E1 -17692.342,E2 -17692.342} C_VEL
LIN {X 0,Y 81.374,Z 749.238,A -85,B 0,C 180,E1 -17686.288,E2 -17686.288} C_VEL
LIN {X 0,Y 86.346,Z 745.866,A -85,B 0,C 180,E1 -17682.892,E2 -17682.892} C_VEL
LIN {X 0,Y 85.24,Z 745.299,A -85,B 0,C 180,E1 -17681.269,E2 -17681.269} C_VEL
LIN {X 0,Y 81.897,Z 744.162,A -85,B 0,C 180,E1 -17676.92,E2 -17676.92} C_VEL
LIN {X 0,Y 78.469,Z 743.389,A -85,B 0,C 180,E1 -17672.505,E2 -17672.505} C_VEL
LIN {X 0,Y 72.738,Z 739.673,A -85,B 0,C 180,E1 -17654.912,E2 -17654.912} C_VEL
LIN {X 0,Y 73.121,Z 737.484,A -85,B 0,C 180,E1 -17645.515,E2 -17645.515} C_VEL
LIN {X 0,Y 83.984,Z 731.214,A -85,B 0,C 180,E1 -17620.443,E2 -17620.443} C_VEL
LIN {X 0,Y 92.542,Z 728.061,A -85,B 0,C 180,E1 -17612.892,E2 -17612.892} C_VEL
LIN {X 0,Y 102.972,Z 724.226,A -85,B 0,C 180,E1 -17606.905,E2 -17606.905} C_VEL
LIN {X 0,Y 101.848,Z 725.659,A -85,B 0,C 180,E1 -17605.908,E2 -17605.908} C_VEL
LIN {X 0,Y 93.964,Z 733.005,A -85,B 0,C 180,E1 -17601.761,E2 -17601.761} C_VEL
LIN {X 0,Y 86.559,Z 739.004,A -85,B 0,C 180,E1 -17596.957,E2 -17596.957} C_VEL
LIN {X 0,Y 79.992,Z 743.838,A -85,B 0,C 180,E1 -17591.227,E2 -17591.227} C_VEL
LIN {X 0,Y 74.213,Z 747.66,A -85,B 0,C 180,E1 -17584.633,E2 -17584.633} C_VEL
LIN {X 0,Y 68.198,Z 751.269,A -85,B 0,C 180,E1 -17574.352,E2 -17574.352} C_VEL
LIN {X 0,Y 64.596,Z 753.387,A -85,B 0,C 180,E1 -17562.576,E2 -17562.576} C_VEL
LIN {X 0,Y 63.338,Z 754.064,A -85,B 0,C 180,E1 -17551.013,E2 -17551.013} C_VEL
LIN {X 0,Y 62.83,Z 754.11,A -85,B 0,C 180,E1 -17545.669,E2 -17545.669} C_VEL
LIN {X 0,Y 61.13,Z 753.697,A -85,B 0,C 180,E1 -17536.626,E2 -17536.626} C_VEL
LIN {X 0,Y 60.584,Z 752.824,A -85,B 0,C 180,E1 -17529.148,E2 -17529.148} C_VEL
LIN {X 0,Y 61.549,Z 751.786,A -85,B 0,C 180,E1 -17523.718,E2 -17523.718} C_VEL
LIN {X 0,Y 62.232,Z 751.36,A -85,B 0,C 180,E1 -17522.038,E2 -17522.038} C_VEL
LIN {X 0,Y 68.506,Z 747.963,A -85,B 0,C 180,E1 -17512.019,E2 -17512.019} C_VEL
LIN {X 0,Y 74.851,Z 744.101,A -85,B 0,C 180,E1 -17505.246,E2 -17505.246} C_VEL
LIN {X 0,Y 81.951,Z 739.23,A -85,B 0,C 180,E1 -17499.492,E2 -17499.492} C_VEL
LIN {X 0,Y 91.138,Z 732.094,A -85,B 0,C 180,E1 -17494.018,E2 -17494.018} C_VEL
LIN {X 0,Y 100.369,Z 723.592,A -85,B 0,C 180,E1 -17489.777,E2 -17489.777} C_VEL
LIN {X 0,Y 108.136,Z 715.061,A -85,B 0,C 180,E1 -17486.679,E2 -17486.679} C_VEL
LIN {X 0,Y 116.4,Z 704.443,A -85,B 0,C 180,E1 -17484.058,E2 -17484.058} C_VEL
LIN {X 0,Y 123.369,Z 693.753,A -85,B 0,C 180,E1 -17482.236,E2 -17482.236} C_VEL
LIN {X 0,Y 129.587,Z 681.988,A -85,B 0,C 180,E1 -17480.699,E2 -17480.699} C_VEL
LIN {X 0,Y 134.291,Z 670.813,A -85,B 0,C 180,E1 -17479.621,E2 -17479.621} C_VEL
LIN {X 0,Y 138.609,Z 657.02,A -85,B 0,C 180,E1 -17478.597,E2 -17478.597} C_VEL
LIN {X 0,Y 141.575,Z 643.262,A -85,B 0,C 180,E1 -17477.962,E2 -17477.962} C_VEL
LIN {X 0,Y 144.535,Z 618.02,A -85,B 0,C 180,E1 -17477.238,E2 -17477.238} C_VEL
LIN {X 0,Y 143.22,Z 613.464,A -85,B 0,C 180,E1 -17474.305,E2 -17474.305} C_VEL
LIN {X 0,Y 142.116,Z 610.079,A -85,B 0,C 180,E1 -17471.229,E2 -17471.229} C_VEL
LIN {X 0,Y 141.251,Z 607.227,A -85,B 0,C 180,E1 -17467.698,E2 -17467.698} C_VEL
LIN {X 0,Y 140.679,Z 605.52,A -85,B 0,C 180,E1 -17462.864,E2 -17462.864} C_VEL
LIN {X 0,Y 140.686,Z 605.699,A -85,B 0,C 180,E1 -17459.643,E2 -17459.643} C_VEL
LIN {X 0,Y 141.232,Z 607.537,A -85,B 0,C 180,E1 -17455.183,E2 -17455.183} C_VEL
LIN {X 0,Y 142.433,Z 611.858,A -85,B 0,C 180,E1 -17450.55,E2 -17450.55} C_VEL
LIN {X 0,Y 143.653,Z 616.093,A -85,B 0,C 180,E1 -17447.383,E2 -17447.383} C_VEL
LIN {X 0,Y 144.474,Z 619.259,A -85,B 0,C 180,E1 -17445.564,E2 -17445.564} C_VEL
LIN {X 0,Y 141.335,Z 645.587,A -85,B 0,C 180,E1 -17444.86,E2 -17444.86} C_VEL
LIN {X 0,Y 138.244,Z 659.734,A -85,B 0,C 180,E1 -17444.294,E2 -17444.294} C_VEL
LIN {X 0,Y 134.183,Z 672.511,A -85,B 0,C 180,E1 -17443.548,E2 -17443.548} C_VEL
LIN {X 0,Y 128.916,Z 685.043,A -85,B 0,C 180,E1 -17442.545,E2 -17442.545} C_VEL
LIN {X 0,Y 122.499,Z 697.099,A -85,B 0,C 180,E1 -17441.182,E2 -17441.182} C_VEL
LIN {X 0,Y 115.369,Z 708.031,A -85,B 0,C 180,E1 -17439.474,E2 -17439.474} C_VEL
LIN {X 0,Y 108.407,Z 717.139,A -85,B 0,C 180,E1 -17437.478,E2 -17437.478} C_VEL
LIN {X 0,Y 100.951,Z 725.663,A -85,B 0,C 180,E1 -17434.815,E2 -17434.815} C_VEL
LIN {X 0,Y 92.219,Z 734.129,A -85,B 0,C 180,E1 -17431.2,E2 -17431.2} C_VEL
LIN {X 0,Y 83.912,Z 741.101,A -85,B 0,C 180,E1 -17426.869,E2 -17426.869} C_VEL
LIN {X 0,Y 76.328,Z 746.835,A -85,B 0,C 180,E1 -17421.492,E2 -17421.492} C_VEL
LIN {X 0,Y 68.002,Z 752.383,A -85,B 0,C 180,E1 -17413.381,E2 -17413.381} C_VEL
LIN {X 0,Y 62.193,Z 756.101,A -85,B 0,C 180,E1 -17404.393,E2 -17404.393} C_VEL
LIN {X 0,Y 57.405,Z 759.157,A -85,B 0,C 180,E1 -17391.538,E2 -17391.538} C_VEL
LIN {X 0,Y 55.711,Z 760.739,A -85,B 0,C 180,E1 -17377.238,E2 -17377.238} C_VEL
LIN {X 0,Y 55.904,Z 760.973,A -85,B 0,C 180,E1 -17369.991,E2 -17369.991} C_VEL
LIN {X 0,Y 55.943,Z 760.77,A -85,B 0,C 180,E1 -17362.774,E2 -17362.774} C_VEL
LIN {X 0,Y 58.111,Z 759.241,A -85,B 0,C 180,E1 -17348.717,E2 -17348.717} C_VEL
LIN {X 0,Y 63.41,Z 756.25,A -85,B 0,C 180,E1 -17336.337,E2 -17336.337} C_VEL
LIN {X 0,Y 69.304,Z 753.001,A -85,B 0,C 180,E1 -17328.755,E2 -17328.755} C_VEL
LIN {X 0,Y 77.706,Z 748.007,A -85,B 0,C 180,E1 -17321.715,E2 -17321.715} C_VEL
LIN {X 0,Y 76.771,Z 747.431,A -85,B 0,C 180,E1 -17319.852,E2 -17319.852} C_VEL
LIN {X 0,Y 70.383,Z 745.661,A -85,B 0,C 180,E1 -17309.951,E2 -17309.951} C_VEL
LIN {X 0,Y 66.404,Z 742.417,A -85,B 0,C 180,E1 -17292.22,E2 -17292.22} C_VEL
LIN {X 0,Y 78.242,Z 735.267,A -85,B 0,C 180,E1 -17258.942,E2 -17258.942} C_VEL
LIN {X 0,Y 90.027,Z 731.424,A -85,B 0,C 180,E1 -17249.183,E2 -17249.183} C_VEL
LIN {X 0,Y 92.354,Z 730.653,A -85,B 0,C 180,E1 -17247.812,E2 -17247.812} C_VEL
LIN {X 0,Y 92.475,Z 731.15,A -85,B 0,C 180,E1 -17246.728,E2 -17246.728} C_VEL
LIN {X 0,Y 84.46,Z 737.565,A -85,B 0,C 180,E1 -17242.242,E2 -17242.242} C_VEL
LIN {X 0,Y 77.112,Z 742.756,A -85,B 0,C 180,E1 -17236.822,E2 -17236.822} C_VEL
LIN {X 0,Y 70.477,Z 746.888,A -85,B 0,C 180,E1 -17230.414,E2 -17230.414} C_VEL
LIN {X 0,Y 64.889,Z 750.064,A -85,B 0,C 180,E1 -17222.798,E2 -17222.798} C_VEL
LIN {X 0,Y 59.428,Z 752.915,A -85,B 0,C 180,E1 -17210.789,E2 -17210.789} C_VEL
LIN {X 0,Y 56.627,Z 754.327,A -85,B 0,C 180,E1 -17197.139,E2 -17197.139} C_VEL
LIN {X 0,Y 56.334,Z 754.426,A -85,B 0,C 180,E1 -17186.437,E2 -17186.437} C_VEL
LIN {X 0,Y 57.703,Z 753.757,A -85,B 0,C 180,E1 -17175.911,E2 -17175.911} C_VEL
LIN {X 0,Y 61.803,Z 751.609,A -85,B 0,C 180,E1 -17162.954,E2 -17162.954} C_VEL
LIN {X 0,Y 62.232,Z 751.36,A -85,B 0,C 180,E1 -17162.038,E2 -17162.038} C_VEL
LIN {X 0,Y 64.174,Z 750.105,A -85,B 0,C 180,E1 -17157.131,E2 -17157.131} C_VEL
LIN {X 0,Y 66.732,Z 747.628,A -85,B 0,C 180,E1 -17149.022,E2 -17149.022} C_VEL
LIN {X 0,Y 69.433,Z 745.23,A -85,B 0,C 180,E1 -17143.05,E2 -17143.05} C_VEL
LIN {X 0,Y 72.427,Z 743.083,A -85,B 0,C 180,E1 -17139.304,E2 -17139.304} C_VEL
LIN {X 0,Y 73.66,Z 742.27,A -85,B 0,C 180,E1 -17138.266,E2 -17138.266} C_VEL
LIN {X 0,Y 83.127,Z 735.79,A -85,B 0,C 180,E1 -17132.292,E2 -17132.292} C_VEL
LIN {X 0,Y 91.728,Z 728.89,A -85,B 0,C 180,E1 -17128.237,E2 -17128.237} C_VEL
LIN {X 0,Y 100.361,Z 720.701,A -85,B 0,C 180,E1 -17124.846,E2 -17124.846} C_VEL
LIN {X 0,Y 108.231,Z 711.932,A -85,B 0,C 180,E1 -17122.297,E2 -17122.297} C_VEL
LIN {X 0,Y 116.062,Z 701.592,A -85,B 0,C 180,E1 -17120.199,E2 -17120.199} C_VEL
LIN {X 0,Y 123.259,Z 690.123,A -85,B 0,C 180,E1 -17118.586,E2 -17118.586} C_VEL
LIN {X 0,Y 128.845,Z 679.042,A -85,B 0,C 180,E1 -17117.355,E2 -17117.355} C_VEL
LIN {X 0,Y 133.895,Z 666.385,A -85,B 0,C 180,E1 -17116.36,E2 -17116.36} C_VEL
LIN {X 0,Y 137.641,Z 653.547,A -85,B 0,C 180,E1 -17115.573,E2 -17115.573} C_VEL
LIN {X 0,Y 140.238,Z 640.166,A -85,B 0,C 180,E1 -17115.078,E2 -17115.078} C_VEL
LIN {X 0,Y 142.344,Z 621.843,A -85,B 0,C 180,E1 -17114.589,E2 -17114.589} C_VEL
LIN {X 0,Y 141.297,Z 617.963,A -85,B 0,C 180,E1 -17111.602,E2 -17111.602} C_VEL
LIN {X 0,Y 140.231,Z 614.079,A -85,B 0,C 180,E1 -17107.003,E2 -17107.003} C_VEL
LIN {X 0,Y 139.811,Z 612.595,A -85,B 0,C 180,E1 -17102.882,E2 -17102.882} C_VEL
LIN {X 0,Y 139.829,Z 612.925,A -85,B 0,C 180,E1 -17099.28,E2 -17099.28} C_VEL
LIN {X 0,Y 140.237,Z 614.541,A -85,B 0,C 180,E1 -17095.689,E2 -17095.689} C_VEL
LIN {X 0,Y 141.121,Z 618.23,A -85,B 0,C 180,E1 -17091.678,E2 -17091.678} C_VEL
LIN {X 0,Y 142.187,Z 622.69,A -85,B 0,C 180,E1 -17088.417,E2 -17088.417} C_VEL
LIN {X 0,Y 142.253,Z 622.966,A -85,B 0,C 180,E1 -17088.242,E2 -17088.242} C_VEL
LIN {X 0,Y 139.596,Z 644.857,A -85,B 0,C 180,E1 -17087.67,E2 -17087.67} C_VEL
LIN {X 0,Y 136.538,Z 658.817,A -85,B 0,C 180,E1 -17087.173,E2 -17087.173} C_VEL
LIN {X 0,Y 132.345,Z 671.885,A -85,B 0,C 180,E1 -17086.502,E2 -17086.502} C_VEL
LIN {X 0,Y 126.962,Z 684.489,A -85,B 0,C 180,E1 -17085.611,E2 -17085.611} C_VEL
LIN {X 0,Y 120.395,Z 696.61,A -85,B 0,C 180,E1 -17084.385,E2 -17084.385} C_VEL
LIN {X 0,Y 113.072,Z 707.568,A -85,B 0,C 180,E1 -17082.852,E2 -17082.852} C_VEL
LIN {X 0,Y 105.873,Z 716.692,A -85,B 0,C 180,E1 -17081.056,E2 -17081.056} C_VEL
LIN {X 0,Y 98.118,Z 725.227,A -85,B 0,C 180,E1 -17078.601,E2 -17078.601} C_VEL
LIN {X 0,Y 89.001,Z 733.703,A -85,B 0,C 180,E1 -17075.229,E2 -17075.229} C_VEL
LIN {X 0,Y 78.818,Z 741.706,A -85,B 0,C 180,E1 -17070.372,E2 -17070.372} C_VEL
LIN {X 0,Y 69.511,Z 748.068,A -85,B 0,C 180,E1 -17063.97,E2 -17063.97} C_VEL
LIN {X 0,Y 63.474,Z 751.7,A -85,B 0,C 180,E1 -17058.37,E2 -17058.37} C_VEL
LIN {X 0,Y 56.398,Z 755.685,A -85,B 0,C 180,E1 -17048.528,E2 -17048.528} C_VEL
LIN {X 0,Y 50.805,Z 758.744,A -85,B 0,C 180,E1 -17034.507,E2 -17034.507} C_VEL
LIN {X 0,Y 48.632,Z 760.327,A -85,B 0,C 180,E1 -17018.298,E2 -17018.298} C_VEL
LIN {X 0,Y 48.791,Z 760.562,A -85,B 0,C 180,E1 -17009.989,E2 -17009.989} C_VEL
LIN {X 0,Y 48.914,Z 760.361,A -85,B 0,C 180,E1 -17001.728,E2 -17001.728} C_VEL
LIN {X 0,Y 51.534,Z 758.83,A -85,B 0,C 180,E1 -16985.839,E2 -16985.839} C_VEL
LIN {X 0,Y 57.624,Z 755.84,A -85,B 0,C 180,E1 -16972.413,E2 -16972.413} C_VEL
LIN {X 0,Y 64.143,Z 752.591,A -85,B 0,C 180,E1 -16964.575,E2 -16964.575} C_VEL
LIN {X 0,Y 68.057,Z 750.52,A -85,B 0,C 180,E1 -16961.181,E2 -16961.181} C_VEL
LIN {X 0,Y 68.623,Z 749.686,A -85,B 0,C 180,E1 -16959.327,E2 -16959.327} C_VEL
LIN {X 0,Y 60.711,Z 746.724,A -85,B 0,C 180,E1 -16940.32,E2 -16940.32} C_VEL
LIN {X 0,Y 72.388,Z 738.987,A -85,B 0,C 180,E1 -16897.147,E2 -16897.147} C_VEL
LIN {X 0,Y 82.621,Z 736.043,A -85,B 0,C 180,E1 -16888.291,E2 -16888.291} C_VEL
LIN {X 0,Y 83.102,Z 735.99,A -85,B 0,C 180,E1 -16887.758,E2 -16887.758} C_VEL
LIN {X 0,Y 74.981,Z 741.583,A -85,B 0,C 180,E1 -16882.828,E2 -16882.828} C_VEL
LIN {X 0,Y 67.553,Z 746.058,A -85,B 0,C 180,E1 -16876.751,E2 -16876.751} C_VEL
LIN {X 0,Y 63.069,Z 748.477,A -85,B 0,C 180,E1 -16871.969,E2 -16871.969} C_VEL
LIN {X 0,Y 55.608,Z 752.084,A -85,B 0,C 180,E1 -16860.378,E2 -16860.378} C_VEL
LIN {X 0,Y 50.858,Z 754.204,A -85,B 0,C 180,E1 -16846.055,E2 -16846.055} C_VEL
LIN {X 0,Y 49.197,Z 754.908,A -85,B 0,C 180,E1 -16830.011,E2 -16830.011} C_VEL
LIN {X 0,Y 50.853,Z 754.167,A -85,B 0,C 180,E1 -16813.965,E2 -16813.965} C_VEL
LIN {X 0,Y 55.597,Z 752.019,A -85,B 0,C 180,E1 -16799.637,E2 -16799.637} C_VEL
LIN {X 0,Y 63.08,Z 748.372,A -85,B 0,C 180,E1 -16788.061,E2 -16788.061} C_VEL
LIN {X 0,Y 69.994,Z 744.514,A -85,B 0,C 180,E1 -16781.156,E2 -16781.156} C_VEL
LIN {X 0,Y 73.66,Z 742.27,A -85,B 0,C 180,E1 -16778.266,E2 -16778.266} C_VEL
LIN {X 0,Y 77.159,Z 739.799,A -85,B 0,C 180,E1 -16775.166,E2 -16775.166} C_VEL
LIN {X 0,Y 82.08,Z 735.461,A -85,B 0,C 180,E1 -16769.805,E2 -16769.805} C_VEL
LIN {X 0,Y 87.322,Z 730.54,A -85,B 0,C 180,E1 -16765.19,E2 -16765.19} C_VEL
LIN {X 0,Y 91.122,Z 727.133,A -85,B 0,C 180,E1 -16763.272,E2 -16763.272} C_VEL
LIN {X 0,Y 99.414,Z 719.272,A -85,B 0,C 180,E1 -16760.512,E2 -16760.512} C_VEL
LIN {X 0,Y 107.359,Z 710.449,A -85,B 0,C 180,E1 -16758.357,E2 -16758.357} C_VEL
LIN {X 0,Y 115.455,Z 699.73,A -85,B 0,C 180,E1 -16756.535,E2 -16756.535} C_VEL
LIN {X 0,Y 122.005,Z 689.21,A -85,B 0,C 180,E1 -16755.25,E2 -16755.25} C_VEL
LIN {X 0,Y 127.742,Z 677.834,A -85,B 0,C 180,E1 -16754.164,E2 -16754.164} C_VEL
LIN {X 0,Y 132.546,Z 665.731,A -85,B 0,C 180,E1 -16753.339,E2 -16753.339} C_VEL
LIN {X 0,Y 136.241,Z 652.974,A -85,B 0,C 180,E1 -16752.642,E2 -16752.642} C_VEL
LIN {X 0,Y 138.782,Z 639.861,A -85,B 0,C 180,E1 -16752.221,E2 -16752.221} C_VEL
LIN {X 0,Y 140.424,Z 626.008,A -85,B 0,C 180,E1 -16751.861,E2 -16751.861} C_VEL
LIN {X 0,Y 139.693,Z 623.057,A -85,B 0,C 180,E1 -16749.046,E2 -16749.046} C_VEL
LIN {X 0,Y 139.232,Z 620.916,A -85,B 0,C 180,E1 -16746.284,E2 -16746.284} C_VEL
LIN {X 0,Y 138.944,Z 619.669,A -85,B 0,C 180,E1 -16742.9,E2 -16742.9} C_VEL
LIN {X 0,Y 138.953,Z 620.064,A -85,B 0,C 180,E1 -16739.276,E2 -16739.276} C_VEL
LIN {X 0,Y 139.231,Z 621.399,A -85,B 0,C 180,E1 -16736.383,E2 -16736.383} C_VEL
LIN {X 0,Y 139.896,Z 624.815,A -85,B 0,C 180,E1 -16732.695,E2 -16732.695} C_VEL
LIN {X 0,Y 140.355,Z 627.075,A -85,B 0,C 180,E1 -16730.911,E2 -16730.911} C_VEL
LIN {X 0,Y 137.695,Z 646.834,A -85,B 0,C 180,E1 -16730.488,E2 -16730.488} C_VEL
LIN {X 0,Y 134.489,Z 660.396,A -85,B 0,C 180,E1 -16730.032,E2 -16730.032} C_VEL
LIN {X 0,Y 130.318,Z 672.726,A -85,B 0,C 180,E1 -16729.462,E2 -16729.462} C_VEL
LIN {X 0,Y 124.543,Z 685.635,A -85,B 0,C 180,E1 -16728.635,E2 -16728.635} C_VEL
LIN {X 0,Y 117.838,Z 697.419,A -85,B 0,C 180,E1 -16727.565,E2 -16727.565} C_VEL
LIN {X 0,Y 109.523,Z 709.259,A -85,B 0,C 180,E1 -16726.039,E2 -16726.039} C_VEL
LIN {X 0,Y 100.706,Z 719.645,A -85,B 0,C 180,E1 -16724.03,E2 -16724.03} C_VEL
LIN {X 0,Y 92.55,Z 727.799,A -85,B 0,C 180,E1 -16721.643,E2 -16721.643} C_VEL
LIN {X 0,Y 83.135,Z 735.772,A -85,B 0,C 180,E1 -16718.402,E2 -16718.402} C_VEL
LIN {X 0,Y 74.065,Z 742.309,A -85,B 0,C 180,E1 -16714.332,E2 -16714.332} C_VEL
LIN {X 0,Y 65.56,Z 747.65,A -85,B 0,C 180,E1 -16709.031,E2 -16709.031} C_VEL
LIN {X 0,Y 58.371,Z 751.589,A -85,B 0,C 180,E1 -16702.987,E2 -16702.987} C_VEL
LIN {X 0,Y 50.97,Z 755.269,A -85,B 0,C 180,E1 -16693.57,E2 -16693.57} C_VEL
LIN {X 0,Y 44.393,Z 758.331,A -85,B 0,C 180,E1 -16678.342,E2 -16678.342} C_VEL
LIN {X 0,Y 41.595,Z 759.915,A -85,B 0,C 180,E1 -16659.715,E2 -16659.715} C_VEL
LIN {X 0,Y 41.687,Z 760.152,A -85,B 0,C 180,E1 -16649.987,E2 -16649.987} C_VEL
LIN {X 0,Y 41.892,Z 759.951,A -85,B 0,C 180,E1 -16640.33,E2 -16640.33} C_VEL
LIN {X 0,Y 45.135,Z 758.42,A -85,B 0,C 180,E1 -16622.139,E2 -16622.139} C_VEL
LIN {X 0,Y 52.169,Z 755.43,A -85,B 0,C 180,E1 -16607.643,E2 -16607.643} C_VEL
LIN {X 0,Y 58.809,Z 752.46,A -85,B 0,C 180,E1 -16600.205,E2 -16600.205} C_VEL
LIN {X 0,Y 59.871,Z 751.489,A -85,B 0,C 180,E1 -16597.625,E2 -16597.625} C_VEL
LIN {X 0,Y 53.542,Z 748.56,A -85,B 0,C 180,E1 -16575.219,E2 -16575.219} C_VEL
LIN {X 0,Y 71.061,Z 741.164,A -85,B 0,C 180,E1 -16530.362,E2 -16530.362} C_VEL
LIN {X 0,Y 72.146,Z 740.896,A -85,B 0,C 180,E1 -16529.415,E2 -16529.415} C_VEL
LIN {X 0,Y 70.327,Z 742.332,A -85,B 0,C 180,E1 -16527.026,E2 -16527.026} C_VEL
LIN {X 0,Y 60.391,Z 747.706,A -85,B 0,C 180,E1 -16519.164,E2 -16519.164} C_VEL
LIN {X 0,Y 53.517,Z 750.881,A -85,B 0,C 180,E1 -16511.055,E2 -16511.055} C_VEL
LIN {X 0,Y 46.445,Z 753.732,A -85,B 0,C 180,E1 -16497.01,E2 -16497.01} C_VEL
LIN {X 0,Y 42.61,Z 755.144,A -85,B 0,C 180,E1 -16479.506,E2 -16479.506} C_VEL
LIN {X 0,Y 42.132,Z 755.316,A -85,B 0,C 180,E1 -16470.012,E2 -16470.012} C_VEL
LIN {X 0,Y 44.089,Z 754.576,A -85,B 0,C 180,E1 -16451.422,E2 -16451.422} C_VEL
LIN {X 0,Y 49.609,Z 752.429,A -85,B 0,C 180,E1 -16435.494,E2 -16435.494} C_VEL
LIN {X 0,Y 57.99,Z 748.783,A -85,B 0,C 180,E1 -16423.365,E2 -16423.365} C_VEL
LIN {X 0,Y 65.549,Z 744.926,A -85,B 0,C 180,E1 -16416.488,E2 -16416.488} C_VEL
LIN {X 0,Y 73.745,Z 740.063,A -85,B 0,C 180,E1 -16410.954,E2 -16410.954} C_VEL
LIN {X 0,Y 84.043,Z 732.932,A -85,B 0,C 180,E1 -16405.994,E2 -16405.994} C_VEL
LIN {X 0,Y 91.122,Z 727.133,A -85,B 0,C 180,E1 -16403.272,E2 -16403.272} C_VEL
LIN {X 0,Y 94.89,Z 723.568,A -85,B 0,C 180,E1 -16401.535,E2 -16401.535} C_VEL
LIN {X 0,Y 100.221,Z 717.56,A -85,B 0,C 180,E1 -16398.117,E2 -16398.117} C_VEL
LIN {X 0,Y 105.409,Z 711.056,A -85,B 0,C 180,E1 -16395.123,E2 -16395.123} C_VEL
LIN {X 0,Y 108.797,Z 706.702,A -85,B 0,C 180,E1 -16394.006,E2 -16394.006} C_VEL
LIN {X 0,Y 116.153,Z 696.5,A -85,B 0,C 180,E1 -16392.689,E2 -16392.689} C_VEL
LIN {X 0,Y 122.846,Z 685.15,A -85,B 0,C 180,E1 -16391.583,E2 -16391.583} C_VEL
LIN {X 0,Y 128.731,Z 672.575,A -85,B 0,C 180,E1 -16390.698,E2 -16390.698} C_VEL
LIN {X 0,Y 133.101,Z 660.204,A -85,B 0,C 180,E1 -16389.98,E2 -16389.98} C_VEL
LIN {X 0,Y 136.392,Z 647.08,A -85,B 0,C 180,E1 -16389.507,E2 -16389.507} C_VEL
LIN {X 0,Y 138.702,Z 631.431,A -85,B 0,C 180,E1 -16389.137,E2 -16389.137} C_VEL
LIN {X 0,Y 138.775,Z 630.423,A -85,B 0,C 180,E1 -16388.983,E2 -16388.983} C_VEL
LIN {X 0,Y 138.256,Z 627.746,A -85,B 0,C 180,E1 -16385.561,E2 -16385.561} C_VEL
LIN {X 0,Y 138.074,Z 626.764,A -85,B 0,C 180,E1 -16382.918,E2 -16382.918} C_VEL
LIN {X 0,Y 138.079,Z 627.185,A -85,B 0,C 180,E1 -16379.271,E2 -16379.271} C_VEL
LIN {X 0,Y 138.246,Z 628.262,A -85,B 0,C 180,E1 -16377.086,E2 -16377.086} C_VEL
LIN {X 0,Y 138.718,Z 631.371,A -85,B 0,C 180,E1 -16373.733,E2 -16373.733} C_VEL
LIN {X 0,Y 136.333,Z 647.782,A -85,B 0,C 180,E1 -16373.385,E2 -16373.385} C_VEL
LIN {X 0,Y 132.985,Z 661.272,A -85,B 0,C 180,E1 -16372.981,E2 -16372.981} C_VEL
LIN {X 0,Y 128.321,Z 674.294,A -85,B 0,C 180,E1 -16372.477,E2 -16372.477} C_VEL
LIN {X 0,Y 122.484,Z 686.697,A -85,B 0,C 180,E1 -16371.771,E2 -16371.771} C_VEL
LIN {X 0,Y 115.659,Z 698.227,A -85,B 0,C 180,E1 -16370.872,E2 -16370.872} C_VEL
LIN {X 0,Y 107.179,Z 709.869,A -85,B 0,C 180,E1 -16369.576,E2 -16369.576} C_VEL
LIN {X 0,Y 98.754,Z 719.439,A -85,B 0,C 180,E1 -16367.96,E2 -16367.96} C_VEL
LIN {X 0,Y 88.906,Z 728.809,A -85,B 0,C 180,E1 -16365.522,E2 -16365.522} C_VEL
LIN {X 0,Y 79.173,Z 736.516,A -85,B 0,C 180,E1 -16362.578,E2 -16362.578} C_VEL
LIN {X 0,Y 71.248,Z 741.886,A -85,B 0,C 180,E1 -16359.546,E2 -16359.546} C_VEL
LIN {X 0,Y 62.177,Z 747.231,A -85,B 0,C 180,E1 -16354.703,E2 -16354.703} C_VEL
LIN {X 0,Y 53.715,Z 751.479,A -85,B 0,C 180,E1 -16348.444,E2 -16348.444} C_VEL
LIN {X 0,Y 46.032,Z 754.854,A -85,B 0,C 180,E1 -16339.745,E2 -16339.745} C_VEL
LIN {X 0,Y 38.229,Z 757.916,A -85,B 0,C 180,E1 -16323.454,E2 -16323.454} C_VEL
LIN {X 0,Y 34.585,Z 759.503,A -85,B 0,C 180,E1 -16301.709,E2 -16301.709} C_VEL
LIN {X 0,Y 34.576,Z 759.742,A -85,B 0,C 180,E1 -16289.985,E2 -16289.985} C_VEL
LIN {X 0,Y 34.904,Z 759.541,A -85,B 0,C 180,E1 -16278.369,E2 -16278.369} C_VEL
LIN {X 0,Y 38.993,Z 758.011,A -85,B 0,C 180,E1 -16257.253,E2 -16257.253} C_VEL
LIN {X 0,Y 47.161,Z 755.021,A -85,B 0,C 180,E1 -16241.815,E2 -16241.815} C_VEL
LIN {X 0,Y 50.947,Z 753.527,A -85,B 0,C 180,E1 -16237.618,E2 -16237.618} C_VEL
LIN {X 0,Y 50.401,Z 752.771,A -85,B 0,C 180,E1 -16233.194,E2 -16233.194} C_VEL
LIN {X 0,Y 61.742,Z 745.082,A -85,B 0,C 180,E1 -16170.909,E2 -16170.909} C_VEL
LIN {X 0,Y 60.493,Z 746.009,A -85,B 0,C 180,E1 -16168.146,E2 -16168.146} C_VEL
LIN {X 0,Y 53.368,Z 749.295,A -85,B 0,C 180,E1 -16162.213,E2 -16162.213} C_VEL
LIN {X 0,Y 43.955,Z 752.901,A -85,B 0,C 180,E1 -16149.774,E2 -16149.774} C_VEL
LIN {X 0,Y 37.452,Z 755.021,A -85,B 0,C 180,E1 -16132.058,E2 -16132.058} C_VEL
LIN {X 0,Y 35.057,Z 755.724,A -85,B 0,C 180,E1 -16110.015,E2 -16110.015} C_VEL
LIN {X 0,Y 37.446,Z 754.985,A -85,B 0,C 180,E1 -16087.968,E2 -16087.968} C_VEL
LIN {X 0,Y 43.942,Z 752.839,A -85,B 0,C 180,E1 -16070.243,E2 -16070.243} C_VEL
LIN {X 0,Y 53.369,Z 749.194,A -85,B 0,C 180,E1 -16057.821,E2 -16057.821} C_VEL
LIN {X 0,Y 61.603,Z 745.337,A -85,B 0,C 180,E1 -16051.186,E2 -16051.186} C_VEL
LIN {X 0,Y 70.359,Z 740.478,A -85,B 0,C 180,E1 -16045.993,E2 -16045.993} C_VEL
LIN {X 0,Y 81.191,Z 733.351,A -85,B 0,C 180,E1 -16041.5,E2 -16041.5} C_VEL
LIN {X 0,Y 90.729,Z 725.753,A -85,B 0,C 180,E1 -16038.449,E2 -16038.449} C_VEL
LIN {X 0,Y 98.78,Z 718.097,A -85,B 0,C 180,E1 -16036.179,E2 -16036.179} C_VEL
LIN {X 0,Y 107.827,Z 707.946,A -85,B 0,C 180,E1 -16034.203,E2 -16034.203} C_VEL
LIN {X 0,Y 108.797,Z 706.702,A -85,B 0,C 180,E1 -16034.006,E2 -16034.006} C_VEL
LIN {X 0,Y 112.094,Z 702.207,A -85,B 0,C 180,E1 -16033.004,E2 -16033.004} C_VEL
LIN {X 0,Y 116.817,Z 694.691,A -85,B 0,C 180,E1 -16030.76,E2 -16030.76} C_VEL
LIN {X 0,Y 121.135,Z 686.822,A -85,B 0,C 180,E1 -16028.743,E2 -16028.743} C_VEL
LIN {X 0,Y 123.692,Z 681.705,A -85,B 0,C 180,E1 -16028.052,E2 -16028.052} C_VEL
LIN {X 0,Y 129.132,Z 669.312,A -85,B 0,C 180,E1 -16027.385,E2 -16027.385} C_VEL
LIN {X 0,Y 133.42,Z 656.176,A -85,B 0,C 180,E1 -16026.796,E2 -16026.796} C_VEL
LIN {X 0,Y 136.348,Z 643.06,A -85,B 0,C 180,E1 -16026.432,E2 -16026.432} C_VEL
LIN {X 0,Y 137.441,Z 635.574,A -85,B 0,C 180,E1 -16026.283,E2 -16026.283} C_VEL
LIN {X 0,Y 137.246,Z 634.127,A -85,B 0,C 180,E1 -16023.854,E2 -16023.854} C_VEL
LIN {X 0,Y 137.204,Z 633.857,A -85,B 0,C 180,E1 -16022.937,E2 -16022.937} C_VEL
LIN {X 0,Y 137.206,Z 634.289,A -85,B 0,C 180,E1 -16019.267,E2 -16019.267} C_VEL
LIN {X 0,Y 137.293,Z 635.208,A -85,B 0,C 180,E1 -16017.663,E2 -16017.663} C_VEL
LIN {X 0,Y 137.369,Z 636.12,A -85,B 0,C 180,E1 -16016.617,E2 -16016.617} C_VEL
LIN {X 0,Y 135.25,Z 649.099,A -85,B 0,C 180,E1 -16016.328,E2 -16016.328} C_VEL
LIN {X 0,Y 131.518,Z 662.991,A -85,B 0,C 180,E1 -16015.979,E2 -16015.979} C_VEL
LIN {X 0,Y 126.87,Z 675.35,A -85,B 0,C 180,E1 -16015.586,E2 -16015.586} C_VEL
LIN {X 0,Y 120.803,Z 687.759,A -85,B 0,C 180,E1 -16015.004,E2 -16015.004} C_VEL
LIN {X 0,Y 113.88,Z 699.034,A -85,B 0,C 180,E1 -16014.294,E2 -16014.294} C_VEL
LIN {X 0,Y 105.26,Z 710.461,A -85,B 0,C 180,E1 -16013.256,E2 -16013.256} C_VEL
LIN {X 0,Y 95.847,Z 720.642,A -85,B 0,C 180,E1 -16011.79,E2 -16011.79} C_VEL
LIN {X 0,Y 85.704,Z 729.749,A -85,B 0,C 180,E1 -16009.713,E2 -16009.713} C_VEL
LIN {X 0,Y 75.67,Z 737.224,A -85,B 0,C 180,E1 -16007.183,E2 -16007.183} C_VEL
LIN {X 0,Y 65.831,Z 743.356,A -85,B 0,C 180,E1 -16003.878,E2 -16003.878} C_VEL
LIN {X 0,Y 56.341,Z 748.351,A -85,B 0,C 180,E1 -15999.289,E2 -15999.289} C_VEL
LIN {X 0,Y 47.314,Z 752.331,A -85,B 0,C 180,E1 -15993.003,E2 -15993.003} C_VEL
LIN {X 0,Y 36.745,Z 756.16,A -85,B 0,C 180,E1 -15979.89,E2 -15979.89} C_VEL
LIN {X 0,Y 29.353,Z 758.479,A -85,B 0,C 180,E1 -15958.591,E2 -15958.591} C_VEL
LIN {X 0,Y 27.632,Z 759.091,A -85,B 0,C 180,E1 -15944.715,E2 -15944.715} C_VEL
LIN {X 0,Y 27.463,Z 759.332,A -85,B 0,C 180,E1 -15929.981,E2 -15929.981} C_VEL
LIN {X 0,Y 27.963,Z 759.13,A -85,B 0,C 180,E1 -15915.424,E2 -15915.424} C_VEL
LIN {X 0,Y 33.244,Z 757.601,A -85,B 0,C 180,E1 -15890.618,E2 -15890.618} C_VEL
LIN {X 0,Y 42.753,Z 754.612,A -85,B 0,C 180,E1 -15874.701,E2 -15874.701} C_VEL
LIN {X 0,Y 42.112,Z 754.091,A -85,B 0,C 180,E1 -15870.043,E2 -15870.043} C_VEL
LIN {X 0,Y 52.067,Z 748.471,A -85,B 0,C 180,E1 -15812.045,E2 -15812.045} C_VEL
LIN {X 0,Y 50.807,Z 749.125,A -85,B 0,C 180,E1 -15809.92,E2 -15809.92} C_VEL
LIN {X 0,Y 43.837,Z 751.697,A -85,B 0,C 180,E1 -15803.303,E2 -15803.303} C_VEL
LIN {X 0,Y 34.418,Z 754.55,A -85,B 0,C 180,E1 -15787.795,E2 -15787.795} C_VEL
LIN {X 0,Y 28.738,Z 755.961,A -85,B 0,C 180,E1 -15764.174,E2 -15764.174} C_VEL
LIN {X 0,Y 27.97,Z 756.133,A -85,B 0,C 180,E1 -15750.019,E2 -15750.019} C_VEL
LIN {X 0,Y 30.995,Z 755.394,A -85,B 0,C 180,E1 -15723.051,E2 -15723.051} C_VEL
LIN {X 0,Y 38.759,Z 753.248,A -85,B 0,C 180,E1 -15703.526,E2 -15703.526} C_VEL
LIN {X 0,Y 49.344,Z 749.604,A -85,B 0,C 180,E1 -15691.308,E2 -15691.308} C_VEL
LIN {X 0,Y 58.252,Z 745.749,A -85,B 0,C 180,E1 -15685.218,E2 -15685.218} C_VEL
LIN {X 0,Y 67.553,Z 740.893,A -85,B 0,C 180,E1 -15680.58,E2 -15680.58} C_VEL
LIN {X 0,Y 78.873,Z 733.769,A -85,B 0,C 180,E1 -15676.713,E2 -15676.713} C_VEL
LIN {X 0,Y 88.505,Z 726.373,A -85,B 0,C 180,E1 -15674.156,E2 -15674.156} C_VEL
LIN {X 0,Y 97.046,Z 718.533,A -85,B 0,C 180,E1 -15672.162,E2 -15672.162} C_VEL
LIN {X 0,Y 106.314,Z 708.407,A -85,B 0,C 180,E1 -15670.506,E2 -15670.506} C_VEL
LIN {X 0,Y 113.951,Z 698.271,A -85,B 0,C 180,E1 -15669.348,E2 -15669.348} C_VEL
LIN {X 0,Y 120.769,Z 687.248,A -85,B 0,C 180,E1 -15668.424,E2 -15668.424} C_VEL
LIN {X 0,Y 123.692,Z 681.705,A -85,B 0,C 180,E1 -15668.052,E2 -15668.052} C_VEL
LIN {X 0,Y 126.103,Z 676.459,A -85,B 0,C 180,E1 -15667.38,E2 -15667.38} C_VEL
LIN {X 0,Y 129.395,Z 667.933,A -85,B 0,C 180,E1 -15665.558,E2 -15665.558} C_VEL
LIN {X 0,Y 132.21,Z 659.148,A -85,B 0,C 180,E1 -15664.004,E2 -15664.004} C_VEL
LIN {X 0,Y 133.693,Z 653.522,A -85,B 0,C 180,E1 -15663.669,E2 -15663.669} C_VEL
LIN {X 0,Y 136.248,Z 641.063,A -85,B 0,C 180,E1 -15663.379,E2 -15663.379} C_VEL
LIN {X 0,Y 136.215,Z 641.265,A -85,B 0,C 180,E1 -15659.631,E2 -15659.631} C_VEL
LIN {X 0,Y 136.221,Z 641.309,A -85,B 0,C 180,E1 -15659.47,E2 -15659.47} C_VEL
LIN {X 0,Y 133.273,Z 655.346,A -85,B 0,C 180,E1 -15659.215,E2 -15659.215} C_VEL
LIN {X 0,Y 129.258,Z 667.963,A -85,B 0,C 180,E1 -15658.955,E2 -15658.955} C_VEL
LIN {X 0,Y 123.893,Z 680.497,A -85,B 0,C 180,E1 -15658.636,E2 -15658.636} C_VEL
LIN {X 0,Y 116.893,Z 693.194,A -85,B 0,C 180,E1 -15658.116,E2 -15658.116} C_VEL
LIN {X 0,Y 109.026,Z 704.586,A -85,B 0,C 180,E1 -15657.523,E2 -15657.523} C_VEL
LIN {X 0,Y 100.306,Z 714.901,A -85,B 0,C 180,E1 -15656.689,E2 -15656.689} C_VEL
LIN {X 0,Y 90.372,Z 724.574,A -85,B 0,C 180,E1 -15655.373,E2 -15655.373} C_VEL
LIN {X 0,Y 79.561,Z 733.246,A -85,B 0,C 180,E1 -15653.537,E2 -15653.537} C_VEL
LIN {X 0,Y 67.585,Z 741.039,A -85,B 0,C 180,E1 -15651.017,E2 -15651.017} C_VEL
LIN {X 0,Y 57.525,Z 746.391,A -85,B 0,C 180,E1 -15647.747,E2 -15647.747} C_VEL
LIN {X 0,Y 46.01,Z 751.355,A -85,B 0,C 180,E1 -15642.213,E2 -15642.213} C_VEL
LIN {X 0,Y 38.361,Z 754.025,A -85,B 0,C 180,E1 -15636.318,E2 -15636.318} C_VEL
LIN {X 0,Y 27.424,Z 757.087,A -85,B 0,C 180,E1 -15620.217,E2 -15620.217} C_VEL
LIN {X 0,Y 20.794,Z 758.678,A -85,B 0,C 180,E1 -15589.727,E2 -15589.727} C_VEL
LIN {X 0,Y 20.343,Z 758.921,A -85,B 0,C 180,E1 -15569.974,E2 -15569.974} C_VEL
LIN {X 0,Y 21.158,Z 758.72,A -85,B 0,C 180,E1 -15550.574,E2 -15550.574} C_VEL
LIN {X 0,Y 28.112,Z 757.191,A -85,B 0,C 180,E1 -15521.383,E2 -15521.383} C_VEL
LIN {X 0,Y 33.329,Z 755.883,A -85,B 0,C 180,E1 -15512.464,E2 -15512.464} C_VEL
LIN {X 0,Y 34.383,Z 755.289,A -85,B 0,C 180,E1 -15507.681,E2 -15507.681} C_VEL
LIN {X 0,Y 41.733,Z 751.496,A -85,B 0,C 180,E1 -15454.699,E2 -15454.699} C_VEL
LIN {X 0,Y 40.001,Z 752.106,A -85,B 0,C 180,E1 -15451.487,E2 -15451.487} C_VEL
LIN {X 0,Y 29.141,Z 754.959,A -85,B 0,C 180,E1 -15436.37,E2 -15436.37} C_VEL
LIN {X 0,Y 21.933,Z 756.37,A -85,B 0,C 180,E1 -15408.714,E2 -15408.714} C_VEL
LIN {X 0,Y 20.89,Z 756.541,A -85,B 0,C 180,E1 -15390.025,E2 -15390.025} C_VEL
LIN {X 0,Y 24.878,Z 755.804,A -85,B 0,C 180,E1 -15355.624,E2 -15355.624} C_VEL
LIN {X 0,Y 34.271,Z 753.657,A -85,B 0,C 180,E1 -15334.914,E2 -15334.914} C_VEL
LIN {X 0,Y 46.065,Z 750.013,A -85,B 0,C 180,E1 -15323.765,E2 -15323.765} C_VEL
LIN {X 0,Y 55.606,Z 746.16,A -85,B 0,C 180,E1 -15318.604,E2 -15318.604} C_VEL
LIN {X 0,Y 65.4,Z 741.307,A -85,B 0,C 180,E1 -15314.758,E2 -15314.758} C_VEL
LIN {X 0,Y 77.137,Z 734.188,A -85,B 0,C 180,E1 -15311.676,E2 -15311.676} C_VEL
LIN {X 0,Y 87.977,Z 726.024,A -85,B 0,C 180,E1 -15309.383,E2 -15309.383} C_VEL
LIN {X 0,Y 97.518,Z 717.278,A -85,B 0,C 180,E1 -15307.761,E2 -15307.761} C_VEL
LIN {X 0,Y 106.975,Z 706.746,A -85,B 0,C 180,E1 -15306.498,E2 -15306.498} C_VEL
LIN {X 0,Y 114.755,Z 696.184,A -85,B 0,C 180,E1 -15305.667,E2 -15305.667} C_VEL
LIN {X 0,Y 121.673,Z 684.621,A -85,B 0,C 180,E1 -15304.934,E2 -15304.934} C_VEL
LIN {X 0,Y 127.333,Z 672.685,A -85,B 0,C 180,E1 -15304.375,E2 -15304.375} C_VEL
LIN {X 0,Y 132.182,Z 658.98,A -85,B 0,C 180,E1 -15303.83,E2 -15303.83} C_VEL
LIN {X 0,Y 133.693,Z 653.522,A -85,B 0,C 180,E1 -15303.669,E2 -15303.669} C_VEL
LIN {X 0,Y 137.636,Z 653.989,A -85,B 0,C 180,E1 -15303.712,E2 -15303.712} C_VEL
LIN {X 0,Y 137.636,Z 711.207,A -85,B 0,C 180,E1 -15303.712,E2 -15303.712} C_VEL
LIN {X 0,Y 118.04,Z 711.207,A -85,B 0,C 180,E1 -15302.107,E2 -15302.107} C_VEL
LIN {X 0,Y 116.079,Z 709.207,A -85,B 0,C 180,E1 -15301.916,E2 -15301.916} C_VEL
LIN {X 0,Y 116.079,Z 700.428,A -85,B 0,C 180,E1 -15301.916,E2 -15301.916} C_VEL
LIN {X 0,Y 112.523,Z 699.244,A -85,B 0,C 180,E1 -15302.232,E2 -15302.232} C_VEL
LIN {X 0,Y 104.663,Z 709.326,A -85,B 0,C 180,E1 -15302.874,E2 -15302.874} C_VEL
LIN {X 0,Y 95.076,Z 719.405,A -85,B 0,C 180,E1 -15303.793,E2 -15303.793} C_VEL
LIN {X 0,Y 84.667,Z 728.368,A -85,B 0,C 180,E1 -15305.141,E2 -15305.141} C_VEL
LIN {X 0,Y 74.293,Z 735.713,A -85,B 0,C 180,E1 -15306.709,E2 -15306.709} C_VEL
LIN {X 0,Y 63.963,Z 741.722,A -85,B 0,C 180,E1 -15308.612,E2 -15308.612} C_VEL
LIN {X 0,Y 53.768,Z 746.571,A -85,B 0,C 180,E1 -15311.435,E2 -15311.435} C_VEL
LIN {X 0,Y 40.388,Z 751.473,A -85,B 0,C 180,E1 -15316.896,E2 -15316.896} C_VEL
LIN {X 0,Y 30.775,Z 754.065,A -85,B 0,C 180,E1 -15324.054,E2 -15324.054} C_VEL
LIN {X 0,Y 19.454,Z 756.213,A -85,B 0,C 180,E1 -15343.775,E2 -15343.775} C_VEL
LIN {X 0,Y 13.81,Z 756.95,A -85,B 0,C 180,E1 -15390.038,E2 -15390.038} C_VEL
LIN {X 0,Y 19.467,Z 756.247,A -85,B 0,C 180,E1 -15436.262,E2 -15436.262} C_VEL
LIN {X 0,Y 30.792,Z 754.126,A -85,B 0,C 180,E1 -15455.96,E2 -15455.96} C_VEL
LIN {X 0,Y 29.235,Z 754.392,A -85,B 0,C 180,E1 -15466.088,E2 -15466.088} C_VEL
LIN {X 0,Y 26.417,Z 756.065,A -85,B 0,C 180,E1 -15500.477,E2 -15500.477} C_VEL
LIN {X 0,Y 25.551,Z 756.478,A -85,B 0,C 180,E1 -15506.228,E2 -15506.228} C_VEL
LIN {X 0,Y 18.59,Z 757.724,A -85,B 0,C 180,E1 -15520.837,E2 -15520.837} C_VEL
LIN {X 0,Y 14.659,Z 758.31,A -85,B 0,C 180,E1 -15541.311,E2 -15541.311} C_VEL
LIN {X 0,Y 13.214,Z 758.509,A -85,B 0,C 180,E1 -15569.96,E2 -15569.96} C_VEL
LIN {X 0,Y 14.282,Z 758.266,A -85,B 0,C 180,E1 -15599.436,E2 -15599.436} C_VEL
LIN {X 0,Y 23.489,Z 756.672,A -85,B 0,C 180,E1 -15633.793,E2 -15633.793} C_VEL
LIN {X 0,Y 36.085,Z 753.611,A -85,B 0,C 180,E1 -15646.794,E2 -15646.794} C_VEL
LIN {X 0,Y 45.813,Z 750.394,A -85,B 0,C 180,E1 -15651.594,E2 -15651.594} C_VEL
LIN {X 0,Y 56.44,Z 745.972,A -85,B 0,C 180,E1 -15654.879,E2 -15654.879} C_VEL
LIN {X 0,Y 68.586,Z 739.597,A -85,B 0,C 180,E1 -15657.35,E2 -15657.35} C_VEL
LIN {X 0,Y 79.075,Z 732.818,A -85,B 0,C 180,E1 -15658.701,E2 -15658.701} C_VEL
LIN {X 0,Y 89.207,Z 724.882,A -85,B 0,C 180,E1 -15659.832,E2 -15659.832} C_VEL
LIN {X 0,Y 98.388,Z 716.252,A -85,B 0,C 180,E1 -15660.652,E2 -15660.652} C_VEL
LIN {X 0,Y 108.07,Z 705.246,A -85,B 0,C 180,E1 -15661.221,E2 -15661.221} C_VEL
LIN {X 0,Y 112.473,Z 699.35,A -85,B 0,C 180,E1 -15661.441,E2 -15661.441} C_VEL
LIN {X 0,Y 112.523,Z 699.244,A -85,B 0,C 180,E1 -15662.232,E2 -15662.232} C_VEL
LIN {X 0,Y 112.627,Z 701.239,A -85,B 0,C 180,E1 -15663.318,E2 -15663.318} C_VEL
LIN {X 0,Y 112.627,Z 755.258,A -85,B 0,C 180,E1 -15663.318,E2 -15663.318} C_VEL
LIN {X 0,Y 61.046,Z 755.258,A -85,B 0,C 180,E1 -15662.838,E2 -15662.838} C_VEL
LIN {X 0,Y 59.046,Z 753.258,A -85,B 0,C 180,E1 -15662.802,E2 -15662.802} C_VEL
LIN {X 0,Y 59.046,Z 747.333,A -85,B 0,C 180,E1 -15662.802,E2 -15662.802} C_VEL
LIN {X 0,Y 56.305,Z 745.49,A -85,B 0,C 180,E1 -15663.25,E2 -15663.25} C_VEL
LIN {X 0,Y 45.858,Z 749.641,A -85,B 0,C 180,E1 -15665.158,E2 -15665.158} C_VEL
LIN {X 0,Y 35.473,Z 752.849,A -85,B 0,C 180,E1 -15667.97,E2 -15667.97} C_VEL
LIN {X 0,Y 21.888,Z 755.731,A -85,B 0,C 180,E1 -15675.673,E2 -15675.673} C_VEL
LIN {X 0,Y 15.424,Z 756.622,A -85,B 0,C 180,E1 -15684.399,E2 -15684.399} C_VEL
LIN {X 0,Y 6.722,Z 757.359,A -85,B 0,C 180,E1 -15750.078,E2 -15750.078} C_VEL
LIN {X 0,Y 15.441,Z 756.656,A -85,B 0,C 180,E1 -15815.628,E2 -15815.628} C_VEL
LIN {X 0,Y 19.744,Z 756.129,A -85,B 0,C 180,E1 -15822.074,E2 -15822.074} C_VEL
LIN {X 0,Y 21.187,Z 755.919,A -85,B 0,C 180,E1 -15827.373,E2 -15827.373} C_VEL
LIN {X 0,Y 19.631,Z 756.353,A -85,B 0,C 180,E1 -15839.997,E2 -15839.997} C_VEL
LIN {X 0,Y 17.505,Z 756.98,A -85,B 0,C 180,E1 -15855.745,E2 -15855.745} C_VEL
LIN {X 0,Y 9.088,Z 757.9,A -85,B 0,C 180,E1 -15879.257,E2 -15879.257} C_VEL
LIN {X 0,Y 6.106,Z 758.099,A -85,B 0,C 180,E1 -15929.914,E2 -15929.914} C_VEL
LIN {X 0,Y 8.787,Z 757.853,A -85,B 0,C 180,E1 -15983.011,E2 -15983.011} C_VEL
LIN {X 0,Y 21.316,Z 756.258,A -85,B 0,C 180,E1 -16011.366,E2 -16011.366} C_VEL
LIN {X 0,Y 35.147,Z 753.196,A -85,B 0,C 180,E1 -16018.234,E2 -16018.234} C_VEL
LIN {X 0,Y 45.675,Z 749.85,A -85,B 0,C 180,E1 -16020.653,E2 -16020.653} C_VEL
LIN {X 0,Y 56.255,Z 745.552,A -85,B 0,C 180,E1 -16022.184,E2 -16022.184} C_VEL
LIN {X 0,Y 56.305,Z 745.49,A -85,B 0,C 180,E1 -16023.25,E2 -16023.25} C_VEL
LIN {X 0,Y 56.305,Z 745.49,A -85,B 0,C 180,E1 -16023.25,E2 -16023.25}

QRS_NEXT_CUT()

QRS_NEXT()
QRS_HOME()

END
